C01789=1059.160,245.472,-93.198,172.780,33.846,156.300
C01790=1059.154,245.224,-93.170,172.776,33.843,156.299
C01791=1059.148,244.975,-93.142,172.774,33.838,156.298
C01792=1059.142,244.726,-93.114,172.772,33.835,156.298
C01793=1059.135,244.479,-93.085,172.770,33.831,156.297
C01794=1059.129,244.231,-93.057,172.767,33.827,156.296
C01795=1059.123,243.982,-93.029,172.765,33.823,156.295
C01796=1059.117,243.733,-93.001,172.763,33.820,156.295
C01797=1059.111,243.485,-92.973,172.761,33.816,156.294
C01798=1059.105,243.237,-92.945,172.759,33.812,156.293
C01799=1059.099,242.988,-92.917,172.755,33.808,156.292
C01800=1059.092,242.740,-92.889,172.753,33.804,156.292
C01801=1059.087,242.492,-92.861,172.751,33.801,156.291
C01802=1059.080,242.243,-92.834,172.749,33.797,156.290
C01803=1059.074,241.994,-92.805,172.747,33.793,156.290
C01804=1059.068,241.747,-92.778,172.744,33.789,156.289
C01805=1059.061,241.498,-92.750,172.742,33.786,156.288
C01806=1059.056,241.249,-92.722,172.740,33.782,156.287
C01807=1059.049,241.001,-92.694,172.738,33.778,156.287
C01808=1059.043,240.753,-92.667,172.734,33.774,156.286
C01809=1059.037,240.504,-92.639,172.732,33.770,156.285
C01810=1059.030,240.255,-92.612,172.730,33.767,156.285
C01811=1059.024,240.008,-92.584,172.728,33.763,156.284
C01812=1059.018,239.759,-92.556,172.726,33.759,156.283
C01813=1059.012,239.511,-92.528,172.723,33.755,156.282
C01814=1059.006,239.263,-92.501,172.721,33.752,156.282
C01815=1059.000,239.014,-92.472,172.719,33.748,156.281
C01816=1058.993,238.765,-92.445,172.717,33.744,156.280
C01817=1058.987,238.517,-92.418,172.714,33.740,156.279
C01818=1058.981,238.269,-92.390,172.712,33.737,156.279
C01819=1058.975,238.020,-92.362,172.709,33.733,156.278
C01820=1058.969,237.772,-92.335,172.707,33.729,156.277
C01821=1058.962,237.523,-92.308,172.705,33.725,156.276
C01822=1058.956,237.275,-92.280,172.703,33.721,156.276
C01823=1058.950,237.027,-92.252,172.701,33.718,156.275
C01824=1058.944,236.778,-92.225,172.699,33.714,156.274
C01825=1058.938,236.530,-92.198,172.696,33.710,156.274
C01826=1058.932,236.297,-92.171,172.694,33.707,156.273
C01827=1058.926,236.065,-92.146,172.691,33.703,156.272
C01828=1058.920,235.833,-92.121,172.689,33.700,156.272
C01829=1058.915,235.599,-92.094,172.687,33.696,156.271
C01830=1058.909,235.367,-92.069,172.685,33.692,156.270
C01831=1058.903,235.135,-92.043,172.683,33.689,156.270
C01832=1058.897,234.902,-92.017,172.681,33.685,156.269
C01833=1058.892,234.670,-91.992,172.679,33.681,156.268
C01834=1058.885,234.421,-91.964,172.677,33.678,156.267
C01835=1058.880,234.173,-91.937,172.675,33.674,156.267
C01836=1058.873,233.924,-91.910,172.673,33.670,156.266
C01837=1058.867,233.676,-91.883,172.671,33.666,156.265
C01838=1058.861,233.427,-91.855,172.668,33.663,156.265
C01839=1058.855,233.180,-91.827,172.666,33.659,156.264
C01840=1058.849,232.930,-91.800,172.664,33.655,156.263
C01841=1058.843,232.683,-91.773,172.661,33.651,156.262
C01842=1058.836,232.434,-91.746,172.659,33.647,156.262
C01843=1058.830,232.185,-91.719,172.657,33.644,156.261
C01844=1058.824,231.937,-91.691,172.655,33.639,156.260
C01845=1058.818,231.688,-91.665,172.653,33.636,156.259
C01846=1058.811,231.440,-91.637,172.651,33.632,156.259
C01847=1058.806,231.192,-91.610,172.649,33.629,156.258
C01848=1058.800,230.943,-91.582,172.647,33.624,156.257
C01849=1058.794,230.695,-91.555,172.644,33.621,156.256
C01850=1058.787,230.445,-91.528,172.641,33.617,156.256
C01851=1058.781,230.198,-91.501,172.639,33.613,156.255
C01852=1058.775,229.949,-91.474,172.637,33.609,156.254
C01853=1058.769,229.701,-91.447,172.635,33.605,156.254
C01854=1058.763,229.452,-91.420,172.633,33.601,156.253
C01855=1058.757,229.204,-91.393,172.631,33.598,156.252
C01856=1058.750,228.954,-91.366,172.629,33.594,156.251
C01857=1058.744,228.707,-91.339,172.627,33.590,156.251
C01858=1058.737,228.458,-91.312,172.625,33.587,156.250
C01859=1058.731,228.210,-91.286,172.623,33.582,156.249
C01860=1058.725,227.961,-91.258,172.620,33.579,156.248
C01861=1058.719,227.713,-91.231,172.617,33.575,156.248
C01862=1058.713,227.464,-91.205,172.615,33.571,156.247
C01863=1058.707,227.215,-91.178,172.613,33.567,156.246
C01864=1058.700,226.967,-91.152,172.611,33.564,156.246
C01865=1058.694,226.719,-91.124,172.609,33.560,156.245
C01866=1058.688,226.471,-91.097,172.607,33.556,156.244
C01867=1058.681,226.221,-91.070,172.605,33.552,156.243
C01868=1058.676,225.973,-91.043,172.603,33.548,156.243
C01869=1058.670,225.725,-91.017,172.601,33.545,156.242
C01870=1058.663,225.476,-90.990,172.599,33.540,156.241
C01871=1058.657,225.228,-90.963,172.597,33.537,156.241
C01872=1058.650,224.979,-90.936,172.595,33.533,156.240
C01873=1058.645,224.731,-90.909,172.592,33.529,156.239
C01874=1058.639,224.483,-90.883,172.590,33.525,156.238
C01875=1058.632,224.233,-90.856,172.588,33.522,156.238
C01876=1058.626,223.985,-90.830,172.586,33.517,156.237
C01877=1058.620,223.737,-90.803,172.584,33.514,156.236
C01878=1058.614,223.488,-90.776,172.582,33.510,156.235
C01879=1058.608,223.240,-90.749,172.580,33.506,156.235
C01880=1058.602,222.991,-90.723,172.578,33.502,156.234
C01881=1058.595,222.743,-90.696,172.576,33.499,156.233
C01882=1058.590,222.506,-90.670,172.574,33.495,156.233
C01883=1058.584,222.270,-90.646,172.572,33.491,156.232
C01884=1058.578,222.033,-90.620,172.570,33.488,156.231
C01885=1058.572,221.797,-90.595,172.568,33.484,156.230
C01886=1058.566,221.561,-90.570,172.565,33.480,156.230
C01887=1058.561,221.324,-90.544,172.563,33.476,156.229
C01888=1058.555,221.088,-90.519,172.561,33.472,156.228
C01889=1058.549,220.852,-90.493,172.559,33.469,156.228
C01890=1058.543,220.603,-90.468,172.557,33.465,156.227
C01891=1058.537,220.354,-90.441,172.555,33.461,156.226
C01892=1058.530,220.106,-90.415,172.553,33.458,156.225
C01893=1058.524,219.857,-90.388,172.551,33.453,156.225
C01894=1058.517,219.609,-90.362,172.549,33.450,156.224
C01895=1058.511,219.360,-90.335,172.547,33.446,156.223
C01896=1058.505,219.112,-90.309,172.545,33.442,156.222
C01897=1058.499,218.863,-90.283,172.543,33.438,156.222
C01898=1058.493,218.614,-90.256,172.541,33.435,156.221
C01899=1058.486,218.366,-90.230,172.539,33.430,156.220
C01900=1058.481,218.118,-90.203,172.537,33.427,156.220
C01901=1058.474,217.868,-90.177,172.535,33.423,156.219
C01902=1058.468,217.620,-90.151,172.532,33.419,156.218
C01903=1058.462,217.372,-90.125,172.530,33.415,156.217
C01904=1058.456,217.124,-90.098,172.528,33.411,156.217
C01905=1058.449,216.874,-90.072,172.526,33.407,156.216
C01906=1058.443,216.626,-90.046,172.524,33.404,156.215
C01907=1058.437,216.378,-90.020,172.522,33.400,156.215
C01908=1058.431,216.129,-89.993,172.520,33.396,156.214
C01909=1058.424,215.880,-89.967,172.519,33.392,156.213
C01910=1058.418,215.632,-89.941,172.517,33.388,156.212
C01911=1058.412,215.384,-89.915,172.515,33.384,156.212
C01912=1058.406,215.135,-89.889,172.513,33.380,156.211
C01913=1058.400,214.887,-89.863,172.511,33.376,156.210
C01914=1058.394,214.637,-89.836,172.509,33.373,156.209
C01915=1058.387,214.389,-89.810,172.507,33.368,156.209
C01916=1058.382,214.141,-89.784,172.505,33.365,156.208
C01917=1058.375,213.892,-89.758,172.503,33.361,156.207
C01918=1058.370,213.644,-89.732,172.500,33.357,156.206
C01919=1058.363,213.395,-89.706,172.498,33.353,156.206
C01920=1058.358,213.147,-89.680,172.496,33.349,156.205
C01921=1058.350,212.898,-89.653,172.494,33.345,156.204
C01922=1058.345,212.649,-89.627,172.492,33.341,156.203
C01923=1058.338,212.401,-89.601,172.490,33.337,156.203
C01924=1058.333,212.152,-89.575,172.488,33.334,156.202
C01925=1058.327,211.904,-89.549,172.486,33.329,156.201
C01926=1058.320,211.655,-89.524,172.485,33.326,156.200
C01927=1058.314,211.405,-89.498,172.483,33.321,156.200
C01928=1058.308,211.157,-89.472,172.481,33.318,156.199
C01929=1058.302,210.909,-89.446,172.479,33.313,156.198
C01930=1058.296,210.660,-89.420,172.477,33.310,156.197
C01931=1058.290,210.412,-89.394,172.475,33.306,156.197
C01932=1058.283,210.164,-89.368,172.473,33.302,156.196
C01933=1058.277,209.915,-89.343,172.471,33.298,156.195
C01934=1058.271,209.666,-89.317,172.469,33.294,156.194
C01935=1058.265,209.418,-89.291,172.467,33.290,156.194
C01936=1058.258,209.168,-89.265,172.465,33.287,156.193
C01937=1058.252,208.920,-89.239,172.463,33.282,156.192
C01938=1058.246,208.686,-89.215,172.461,33.279,156.192
C01939=1058.241,208.453,-89.191,172.459,33.275,156.191
C01940=1058.234,208.219,-89.167,172.457,33.271,156.190
C01941=1058.229,207.985,-89.143,172.455,33.268,156.190
C01942=1058.223,207.751,-89.119,172.454,33.264,156.189
C01943=1058.217,207.517,-89.094,172.452,33.260,156.188
C01944=1058.212,207.283,-89.070,172.450,33.257,156.187
C01945=1058.206,207.049,-89.046,172.448,33.253,156.187
C01946=1058.180,205.999,-88.941,172.259,33.165,156.176
C01947=1058.174,205.751,-88.916,172.256,33.162,156.175
C01948=1058.169,205.502,-88.892,172.254,33.159,156.175
C01949=1058.163,205.253,-88.867,172.252,33.156,156.174
C01950=1058.157,205.005,-88.843,172.249,33.153,156.173
C01951=1058.151,204.756,-88.818,172.247,33.150,156.173
C01952=1058.145,204.507,-88.793,172.245,33.147,156.172
C01953=1058.139,204.259,-88.768,172.242,33.144,156.172
C01954=1058.133,204.010,-88.743,172.240,33.140,156.171
C01955=1058.128,203.761,-88.719,172.238,33.138,156.171
C01956=1058.122,203.512,-88.694,172.235,33.135,156.170
C01957=1058.116,203.263,-88.669,172.233,33.132,156.170
C01958=1058.110,203.015,-88.645,172.231,33.128,156.169
C01959=1058.104,202.766,-88.621,172.228,33.125,156.169
C01960=1058.098,202.518,-88.596,172.225,33.122,156.168
C01961=1058.092,202.268,-88.571,172.223,33.120,156.168
C01962=1058.087,202.020,-88.547,172.220,33.116,156.167
C01963=1058.081,201.771,-88.521,172.218,33.113,156.166
C01964=1058.074,201.522,-88.497,172.216,33.110,156.166
C01965=1058.069,201.274,-88.473,172.213,33.107,156.165
C01966=1058.062,201.025,-88.449,172.211,33.104,156.165
C01967=1058.057,200.777,-88.424,172.209,33.101,156.164
C01968=1058.050,200.528,-88.400,172.207,33.099,156.164
C01969=1058.044,200.278,-88.375,172.204,33.095,156.163
C01970=1058.039,200.030,-88.351,172.202,33.093,156.163
C01971=1058.032,199.781,-88.327,172.200,33.090,156.162
C01972=1058.026,199.533,-88.302,172.197,33.087,156.162
C01973=1058.020,199.284,-88.278,172.195,33.084,156.161
C01974=1058.015,199.035,-88.254,172.193,33.081,156.161
C01975=1058.008,198.786,-88.230,172.190,33.078,156.160
C01976=1058.003,198.538,-88.206,172.188,33.075,156.160
C01977=1057.996,198.289,-88.182,172.186,33.072,156.159
C01978=1057.991,198.040,-88.157,172.184,33.069,156.159
C01979=1057.984,197.792,-88.132,172.181,33.066,156.158
C01980=1057.978,197.543,-88.108,172.179,33.063,156.158
C01981=1057.973,197.294,-88.084,172.177,33.061,156.157
C01982=1057.966,197.045,-88.060,172.174,33.057,156.157
C01983=1057.961,196.796,-88.035,172.172,33.054,156.156
C01984=1057.955,196.548,-88.012,172.170,33.052,156.156
C01985=1057.949,196.299,-87.987,172.168,33.048,156.155
C01986=1057.943,196.051,-87.964,172.166,33.046,156.155
C01987=1057.937,195.801,-87.939,172.164,33.043,156.154
C01988=1057.931,195.553,-87.915,172.162,33.040,156.154
C01989=1057.925,195.304,-87.891,172.160,33.037,156.153
C01990=1057.919,195.055,-87.867,172.157,33.034,156.153
C01991=1057.913,194.806,-87.842,172.155,33.031,156.152
C01992=1057.907,194.558,-87.819,172.153,33.028,156.152
C01993=1057.901,194.309,-87.794,172.151,33.025,156.151
C01994=1057.895,194.060,-87.770,172.148,33.022,156.151
C01995=1057.890,193.812,-87.746,172.146,33.019,156.150
C01996=1057.883,193.562,-87.723,172.144,33.017,156.150
C01997=1057.878,193.314,-87.699,172.142,33.014,156.149
C01998=1057.871,193.065,-87.675,172.140,33.010,156.149
C01999=1057.866,192.816,-87.650,172.137,33.008,156.148
C02000=1057.860,192.568,-87.627,172.135,33.005,156.148
C02001=1057.854,192.318,-87.602,172.133,33.002,156.147
C02002=1057.848,192.070,-87.578,172.131,32.999,156.147
C02003=1057.843,191.821,-87.555,172.128,32.996,156.146
C02004=1057.836,191.572,-87.531,172.126,32.993,156.146
C02005=1057.831,191.323,-87.507,172.124,32.990,156.145
C02006=1057.824,191.074,-87.482,172.122,32.987,156.145
C02007=1057.819,190.791,-87.456,172.119,32.984,156.144
C02008=1057.812,190.507,-87.428,172.117,32.980,156.143
C02009=1057.805,190.223,-87.401,172.114,32.977,156.143
C02010=1057.799,189.940,-87.373,172.112,32.974,156.142
C02011=1057.792,189.691,-87.349,172.110,32.971,156.142
C02012=1057.787,189.442,-87.326,172.107,32.968,156.141
C02013=1057.781,189.193,-87.302,172.105,32.965,156.141
C02014=1057.774,188.944,-87.278,172.103,32.963,156.140
C02015=1057.769,188.695,-87.255,172.101,32.959,156.140
C02016=1057.763,188.447,-87.231,172.099,32.957,156.139
C02017=1057.758,188.198,-87.207,172.096,32.954,156.139
C02018=1057.752,187.949,-87.183,172.094,32.951,156.138
C02019=1057.746,187.700,-87.159,172.092,32.948,156.138
C02020=1057.740,187.452,-87.136,172.090,32.945,156.137
C02021=1057.735,187.203,-87.113,172.088,32.942,156.137
C02022=1057.729,186.954,-87.088,172.086,32.939,156.136
C02023=1057.723,186.705,-87.064,172.083,32.936,156.136
C02024=1057.718,186.456,-87.041,172.081,32.933,156.135
C02025=1057.712,186.208,-87.017,172.079,32.931,156.135
C02026=1057.706,185.958,-86.993,172.077,32.928,156.134
C02027=1057.700,185.710,-86.970,172.075,32.925,156.134
C02028=1057.694,185.461,-86.946,172.073,32.922,156.133
C02029=1057.689,185.212,-86.922,172.071,32.919,156.133
C02030=1057.683,184.964,-86.899,172.068,32.916,156.132
C02031=1057.677,184.714,-86.875,172.066,32.913,156.132
C02032=1057.671,184.466,-86.851,172.064,32.910,156.131
C02033=1057.666,184.217,-86.828,172.062,32.908,156.131
C02034=1057.660,183.969,-86.804,172.060,32.905,156.130
C02035=1057.653,183.719,-86.781,172.058,32.902,156.130
C02036=1057.647,183.470,-86.758,172.055,32.899,156.129
C02037=1057.641,183.222,-86.735,172.053,32.897,156.129
C02038=1057.635,182.972,-86.711,172.051,32.894,156.128
C02039=1057.629,182.724,-86.688,172.049,32.891,156.128
C02040=1057.623,182.475,-86.665,172.047,32.889,156.128
C02041=1057.618,182.226,-86.642,172.045,32.886,156.127
C02042=1057.610,181.977,-86.618,172.042,32.883,156.127
C02043=1057.604,181.729,-86.595,172.040,32.880,156.126
C02044=1057.599,181.480,-86.572,172.038,32.878,156.126
C02045=1057.593,181.231,-86.549,172.036,32.875,156.125
C02046=1057.586,180.982,-86.525,172.034,32.872,156.125
C02047=1057.581,180.733,-86.502,172.032,32.869,156.124
C02048=1057.575,180.485,-86.479,172.030,32.867,156.124
C02049=1057.569,180.236,-86.456,172.027,32.864,156.123
C02050=1057.563,179.986,-86.433,172.025,32.862,156.123
C02051=1057.557,179.737,-86.410,172.023,32.858,156.122
C02052=1057.550,179.489,-86.387,172.021,32.856,156.122
C02053=1057.544,179.240,-86.364,172.019,32.853,156.122
C02054=1057.539,178.991,-86.341,172.017,32.851,156.121
C02055=1057.532,178.742,-86.317,172.015,32.848,156.121
C02056=1057.526,178.494,-86.294,172.013,32.845,156.120
C02057=1057.520,178.245,-86.271,172.011,32.842,156.120
C02058=1057.515,177.996,-86.248,172.009,32.840,156.119
C02059=1057.509,177.747,-86.225,172.007,32.837,156.119
C02060=1057.502,177.498,-86.202,172.005,32.834,156.118
C02061=1057.496,177.249,-86.178,172.003,32.831,156.118
C02062=1057.490,177.000,-86.155,172.001,32.829,156.117
C02063=1057.484,176.752,-86.133,171.999,32.826,156.117
C02064=1057.479,176.503,-86.110,171.997,32.823,156.116
C02065=1057.473,176.254,-86.087,171.995,32.821,156.116
C02066=1057.467,176.005,-86.064,171.993,32.818,156.116
C02067=1057.461,175.756,-86.041,171.990,32.815,156.115
C02068=1057.454,175.507,-86.018,171.988,32.812,156.115
C02069=1057.448,175.258,-85.994,171.986,32.810,156.114
C02070=1057.443,175.009,-85.971,171.984,32.807,156.114
C02071=1057.436,174.725,-85.946,171.982,32.804,156.113
C02072=1057.429,174.441,-85.919,171.979,32.801,156.113
C02073=1057.422,174.156,-85.893,171.977,32.798,156.112
C02074=1057.416,173.872,-85.867,171.975,32.795,156.112
C02075=1057.410,173.623,-85.844,171.973,32.792,156.111
C02076=1057.404,173.374,-85.822,171.971,32.789,156.111
C02077=1057.398,173.125,-85.799,171.968,32.786,156.110
C02078=1057.393,172.876,-85.776,171.966,32.784,156.110
C02079=1057.386,172.628,-85.753,171.964,32.781,156.109
C02080=1057.380,172.379,-85.730,171.962,32.778,156.109
C02081=1057.375,172.130,-85.707,171.960,32.776,156.108
C02082=1057.369,171.881,-85.684,171.958,32.773,156.108
C02083=1057.363,171.632,-85.661,171.956,32.770,156.108
C02084=1057.357,171.384,-85.639,171.954,32.768,156.107
C02085=1057.351,171.135,-85.616,171.952,32.765,156.107
C02086=1057.345,170.886,-85.593,171.950,32.762,156.106
C02087=1057.340,170.637,-85.570,171.948,32.760,156.106
C02088=1057.334,170.388,-85.547,171.946,32.757,156.105
C02089=1057.327,170.139,-85.525,171.944,32.754,156.105
C02090=1057.322,169.891,-85.502,171.942,32.751,156.104
C02091=1057.316,169.641,-85.480,171.940,32.749,156.104
C02092=1057.311,169.392,-85.457,171.939,32.746,156.103
C02093=1057.305,169.143,-85.434,171.937,32.744,156.103
C02094=1057.298,168.895,-85.412,171.935,32.740,156.102
C02095=1057.293,168.646,-85.389,171.933,32.738,156.102
C02096=1057.287,168.397,-85.366,171.931,32.735,156.102
C02097=1057.281,168.147,-85.343,171.929,32.733,156.101
C02098=1057.275,167.899,-85.321,171.927,32.730,156.101
C02099=1057.269,167.650,-85.298,171.925,32.727,156.100
C02100=1057.264,167.402,-85.276,171.923,32.724,156.100
C02101=1057.258,167.153,-85.253,171.921,32.722,156.099
C02102=1057.252,166.904,-85.231,171.919,32.719,156.099
C02103=1057.246,166.655,-85.208,171.917,32.716,156.098
C02104=1057.241,166.406,-85.185,171.915,32.713,156.098
C02105=1057.235,166.157,-85.162,171.913,32.711,156.097
C02106=1057.229,165.908,-85.141,171.911,32.708,156.097
C02107=1057.223,165.659,-85.118,171.909,32.706,156.097
C02108=1057.217,165.410,-85.095,171.907,32.702,156.096
C02109=1057.213,165.161,-85.073,171.905,32.700,156.096
C02110=1057.206,164.913,-85.050,171.903,32.697,156.095
C02111=1057.200,164.664,-85.027,171.901,32.695,156.095
C02112=1057.195,164.414,-85.005,171.899,32.692,156.094
C02113=1057.189,164.165,-84.982,171.897,32.689,156.094
C02114=1057.183,163.917,-84.960,171.895,32.686,156.093
C02115=1057.177,163.667,-84.938,171.893,32.684,156.093
C02116=1057.172,163.419,-84.915,171.891,32.681,156.092
C02117=1057.166,163.170,-84.892,171.889,32.678,156.092
C02118=1057.160,162.921,-84.871,171.887,32.675,156.091
C02119=1057.155,162.672,-84.848,171.885,32.673,156.091
C02120=1057.149,162.422,-84.825,171.884,32.670,156.091
C02121=1057.143,162.175,-84.803,171.882,32.668,156.090
C02122=1057.138,161.926,-84.780,171.880,32.665,156.090
C02123=1057.132,161.676,-84.758,171.878,32.662,156.089
C02124=1057.126,161.427,-84.735,171.876,32.659,156.089
C02125=1057.120,161.178,-84.714,171.874,32.657,156.088
C02126=1057.115,160.930,-84.691,171.872,32.654,156.088
C02127=1057.109,160.681,-84.669,171.870,32.651,156.087
C02128=1057.103,160.432,-84.646,171.868,32.648,156.087
C02129=1057.097,160.182,-84.625,171.866,32.646,156.087
C02130=1057.091,159.934,-84.603,171.864,32.643,156.086
C02131=1057.085,159.684,-84.580,171.862,32.641,156.086
C02132=1057.079,159.435,-84.559,171.860,32.638,156.085
C02133=1057.074,159.187,-84.536,171.858,32.636,156.085
C02134=1057.068,158.938,-84.514,171.856,32.633,156.084
C02135=1057.061,158.653,-84.489,171.854,32.630,156.084
C02136=1057.054,158.368,-84.464,171.852,32.627,156.083
C02137=1057.047,158.084,-84.439,171.849,32.624,156.083
C02138=1057.040,157.799,-84.414,171.847,32.621,156.082
C02139=1057.034,157.550,-84.391,171.845,32.619,156.082
C02140=1057.029,157.302,-84.370,171.843,32.616,156.082
C02141=1057.023,157.052,-84.348,171.841,32.614,156.081
C02142=1057.017,156.804,-84.325,171.839,32.611,156.081
C02143=1057.011,156.554,-84.303,171.837,32.608,156.080
C02144=1057.005,156.305,-84.282,171.836,32.606,156.080
C02145=1056.999,156.057,-84.259,171.835,32.603,156.079
C02146=1056.993,155.808,-84.237,171.833,32.601,156.079
C02147=1056.987,155.559,-84.216,171.831,32.598,156.079
C02148=1056.981,155.310,-84.193,171.829,32.595,156.078
C02149=1056.976,155.061,-84.172,171.827,32.593,156.078
C02150=1056.970,154.812,-84.150,171.825,32.590,156.077
C02151=1056.963,154.563,-84.128,171.823,32.588,156.077
C02152=1056.958,154.314,-84.105,171.821,32.585,156.076
C02153=1056.952,154.065,-84.084,171.819,32.583,156.076
C02154=1056.946,153.816,-84.062,171.817,32.580,156.076
C02155=1056.940,153.567,-84.041,171.815,32.577,156.075
C02156=1056.934,153.318,-84.019,171.813,32.575,156.075
C02157=1056.928,153.069,-83.996,171.811,32.572,156.074
C02158=1056.922,152.820,-83.975,171.809,32.570,156.074
C02159=1056.916,152.571,-83.953,171.807,32.567,156.073
C02160=1056.910,152.322,-83.932,171.805,32.564,156.073
C02161=1056.904,152.073,-83.910,171.804,32.562,156.072
C02162=1056.898,151.824,-83.889,171.802,32.559,156.072
C02163=1056.893,151.575,-83.867,171.800,32.557,156.072
C02164=1056.887,151.325,-83.845,171.798,32.554,156.071
C02165=1056.881,151.078,-83.823,171.796,32.552,156.071
C02166=1056.875,150.828,-83.801,171.795,32.549,156.070
C02167=1056.869,150.579,-83.780,171.793,32.546,156.070
C02168=1056.863,150.331,-83.758,171.791,32.544,156.069
C02169=1056.858,150.081,-83.736,171.789,32.541,156.069
C02170=1056.851,149.832,-83.715,171.787,32.539,156.069
C02171=1056.846,149.583,-83.693,171.785,32.536,156.068
C02172=1056.840,149.334,-83.672,171.784,32.533,156.068
C02173=1056.833,149.085,-83.650,171.782,32.531,156.067
C02174=1056.828,148.836,-83.629,171.780,32.528,156.067
C02175=1056.822,148.587,-83.607,171.778,32.526,156.066
C02176=1056.816,148.338,-83.585,171.776,32.523,156.066
C02177=1056.810,148.090,-83.564,171.774,32.521,156.066
C02178=1056.804,147.840,-83.543,171.772,32.518,156.065
C02179=1056.798,147.591,-83.520,171.770,32.516,156.065
C02180=1056.792,147.343,-83.500,171.768,32.513,156.064
C02181=1056.786,147.093,-83.478,171.766,32.511,156.064
C02182=1056.780,146.844,-83.456,171.765,32.508,156.064
C02183=1056.774,146.596,-83.435,171.763,32.506,156.063
C02184=1056.768,146.347,-83.413,171.761,32.503,156.063
C02185=1056.762,146.097,-83.393,171.759,32.500,156.062
C02186=1056.757,145.848,-83.371,171.758,32.498,156.062
C02187=1056.751,145.599,-83.350,171.756,32.496,156.062
C02188=1056.744,145.350,-83.328,171.754,32.493,156.061
C02189=1056.739,145.101,-83.307,171.752,32.491,156.061
C02190=1056.733,144.852,-83.285,171.750,32.488,156.060
C02191=1056.726,144.603,-83.263,171.748,32.485,156.060
C02192=1056.721,144.354,-83.242,171.747,32.483,156.059
C02193=1056.715,144.105,-83.221,171.745,32.480,156.059
C02194=1056.709,143.856,-83.201,171.743,32.478,156.059
C02195=1056.703,143.607,-83.179,171.741,32.476,156.058
C02196=1056.696,143.358,-83.157,171.739,32.473,156.058
C02197=1056.691,143.109,-83.136,171.737,32.470,156.057
C02198=1056.685,142.860,-83.115,171.735,32.468,156.057
C02199=1056.678,142.575,-83.090,171.733,32.465,156.056
C02200=1056.672,142.290,-83.066,171.731,32.462,156.056
C02201=1056.665,142.005,-83.043,171.729,32.459,156.055
C02202=1056.658,141.720,-83.018,171.727,32.456,156.055
C02203=1056.653,141.472,-82.996,171.725,32.454,156.055
C02204=1056.646,141.222,-82.975,171.724,32.451,156.054
C02205=1056.640,140.973,-82.954,171.722,32.448,156.054
C02206=1056.634,140.724,-82.933,171.720,32.446,156.053
C02207=1056.628,140.475,-82.911,171.719,32.444,156.053
C02208=1056.623,140.226,-82.891,171.717,32.441,156.053
C02209=1056.617,139.977,-82.869,171.715,32.439,156.052
C02210=1056.611,139.728,-82.848,171.713,32.436,156.052
C02211=1056.605,139.478,-82.827,171.711,32.434,156.051
C02212=1056.599,139.230,-82.806,171.709,32.431,156.051
C02213=1056.593,138.981,-82.785,171.707,32.428,156.050
C02214=1056.588,138.732,-82.764,171.706,32.426,156.050
C02215=1056.581,138.483,-82.743,171.704,32.424,156.050
C02216=1056.575,138.234,-82.723,171.702,32.421,156.049
C02217=1056.569,137.985,-82.701,171.700,32.419,156.049
C02218=1056.563,137.735,-82.679,171.698,32.416,156.048
C02219=1056.557,137.487,-82.659,171.696,32.413,156.048
C02220=1056.551,137.237,-82.638,171.695,32.411,156.048
C02221=1056.546,136.988,-82.617,171.693,32.409,156.047
C02222=1056.539,136.739,-82.596,171.692,32.406,156.047
C02223=1056.533,136.490,-82.576,171.690,32.404,156.046
C02224=1056.527,136.241,-82.554,171.688,32.401,156.046
C02225=1056.521,135.992,-82.534,171.686,32.398,156.046
C02226=1056.515,135.743,-82.512,171.684,32.396,156.045
C02227=1056.510,135.494,-82.492,171.683,32.394,156.045
C02228=1056.503,135.245,-82.471,171.681,32.391,156.044
C02229=1056.498,134.996,-82.450,171.679,32.389,156.044
C02230=1056.492,134.747,-82.429,171.677,32.386,156.043
C02231=1056.486,134.498,-82.409,171.675,32.384,156.043
C02232=1056.479,134.249,-82.387,171.673,32.381,156.043
C02233=1056.474,134.000,-82.366,171.672,32.379,156.042
C02234=1056.468,133.751,-82.346,171.670,32.376,156.042
C02235=1056.462,133.502,-82.325,171.668,32.374,156.041
C02236=1056.457,133.252,-82.304,171.666,32.371,156.041
C02237=1056.450,133.004,-82.283,171.664,32.369,156.041
C02238=1056.445,132.754,-82.263,171.664,32.367,156.040
C02239=1056.438,132.506,-82.242,171.662,32.364,156.040
C02240=1056.432,132.256,-82.221,171.660,32.361,156.039
C02241=1056.427,132.007,-82.201,171.658,32.359,156.039
C02242=1056.420,131.758,-82.180,171.656,32.356,156.039
C02243=1056.415,131.509,-82.159,171.654,32.354,156.038
C02244=1056.408,131.260,-82.139,171.653,32.352,156.038
C02245=1056.403,131.011,-82.117,171.651,32.349,156.037
C02246=1056.396,130.762,-82.097,171.649,32.347,156.037
C02247=1056.390,130.513,-82.077,171.647,32.344,156.037
C02248=1056.384,130.264,-82.055,171.645,32.342,156.036
C02249=1056.378,130.015,-82.035,171.644,32.340,156.036
C02250=1056.372,129.765,-82.015,171.642,32.337,156.035
C02251=1056.366,129.516,-81.995,171.640,32.335,156.035
C02252=1056.359,129.267,-81.974,171.638,32.332,156.035
C02253=1056.353,129.019,-81.954,171.636,32.330,156.034
C02254=1056.348,128.769,-81.933,171.635,32.327,156.034
C02255=1056.342,128.520,-81.913,171.634,32.325,156.033
C02256=1056.336,128.271,-81.891,171.632,32.323,156.033
C02257=1056.329,128.022,-81.871,171.630,32.320,156.033
C02258=1056.323,127.773,-81.851,171.628,32.318,156.032
C02259=1056.318,127.523,-81.830,171.626,32.315,156.032
C02260=1056.312,127.274,-81.810,171.625,32.313,156.032
C02261=1056.306,127.026,-81.790,171.623,32.311,156.031
C02262=1056.299,126.776,-81.769,171.621,32.308,156.031
C02263=1056.292,126.492,-81.746,171.619,32.305,156.030
C02264=1056.285,126.207,-81.722,171.617,32.303,156.030
C02265=1056.279,125.922,-81.699,171.615,32.300,156.029
C02266=1056.272,125.636,-81.676,171.613,32.297,156.029
C02267=1056.266,125.388,-81.655,171.611,32.295,156.029
C02268=1056.259,125.138,-81.635,171.609,32.292,156.028
C02269=1056.254,124.889,-81.615,171.608,32.290,156.028
C02270=1056.248,124.640,-81.595,171.607,32.287,156.027
C02271=1056.241,124.391,-81.574,171.605,32.285,156.027
C02272=1056.236,124.142,-81.554,171.603,32.282,156.027
C02273=1056.230,123.893,-81.534,171.601,32.280,156.026
C02274=1056.224,123.643,-81.513,171.600,32.277,156.026
C02275=1056.218,123.395,-81.493,171.598,32.275,156.025
C02276=1056.212,123.145,-81.473,171.596,32.273,156.025
C02277=1056.206,122.896,-81.453,171.594,32.270,156.025
C02278=1056.200,122.647,-81.433,171.592,32.268,156.024
C02279=1056.194,122.398,-81.412,171.591,32.265,156.024
C02280=1056.188,122.148,-81.392,171.589,32.263,156.023
C02281=1056.182,121.900,-81.372,171.587,32.260,156.023
C02282=1056.177,121.651,-81.351,171.585,32.258,156.023
C02283=1056.171,121.402,-81.331,171.585,32.256,156.022
C02284=1056.164,121.152,-81.311,171.583,32.253,156.022
C02285=1056.158,120.903,-81.291,171.581,32.250,156.021
C02286=1056.153,120.654,-81.270,171.579,32.248,156.021
C02287=1056.146,120.405,-81.250,171.577,32.246,156.021
C02288=1056.140,120.156,-81.230,171.576,32.243,156.020
C02289=1056.134,119.907,-81.210,171.574,32.241,156.020
C02290=1056.129,119.658,-81.190,171.572,32.238,156.019
C02291=1056.122,119.408,-81.169,171.570,32.236,156.019
C02292=1056.116,119.160,-81.149,171.569,32.234,156.019
C02293=1056.111,118.911,-81.129,171.567,32.231,156.018
C02294=1056.105,118.662,-81.109,171.565,32.228,156.018
C02295=1056.099,118.412,-81.090,171.563,32.226,156.017
C02296=1056.093,118.163,-81.069,171.562,32.224,156.017
C02297=1056.088,117.914,-81.049,171.561,32.221,156.017
C02298=1056.082,117.665,-81.029,171.559,32.218,156.016
C02299=1056.076,117.416,-81.009,171.557,32.216,156.016
C02300=1056.070,117.167,-80.989,171.556,32.214,156.015
C02301=1056.064,116.917,-80.968,171.554,32.211,156.015
C02302=1056.058,116.668,-80.949,171.552,32.209,156.015
C02303=1056.052,116.419,-80.929,171.550,32.206,156.014
C02304=1056.046,116.170,-80.909,171.549,32.204,156.014
C02305=1056.041,115.921,-80.888,171.547,32.202,156.013
C02306=1056.034,115.672,-80.868,171.545,32.199,156.013
C02307=1056.028,115.422,-80.849,171.543,32.196,156.013
C02308=1056.022,115.173,-80.829,171.542,32.194,156.012
C02309=1056.016,114.925,-80.809,171.540,32.192,156.012
C02310=1056.011,114.676,-80.788,171.538,32.189,156.011
C02311=1056.006,114.426,-80.769,171.538,32.187,156.011
C02312=1056.000,114.177,-80.749,171.536,32.184,156.011
C02313=1055.993,113.928,-80.729,171.534,32.181,156.010
C02314=1055.987,113.679,-80.709,171.532,32.179,156.010
C02315=1055.981,113.430,-80.689,171.531,32.177,156.009
C02316=1055.975,113.181,-80.670,171.529,32.174,156.009
C02317=1055.969,112.932,-80.650,171.527,32.172,156.009
C02318=1055.963,112.682,-80.630,171.525,32.169,156.008
C02319=1055.957,112.433,-80.610,171.524,32.167,156.008
C02320=1055.951,112.184,-80.590,171.522,32.165,156.008
C02321=1055.945,111.935,-80.571,171.520,32.162,156.007
C02322=1055.939,111.686,-80.551,171.518,32.160,156.007
C02323=1055.933,111.437,-80.531,171.517,32.158,156.006
C02324=1055.927,111.187,-80.511,171.516,32.155,156.006
C02325=1055.921,110.938,-80.491,171.514,32.153,156.006
C02326=1055.915,110.689,-80.472,171.512,32.150,156.005
C02327=1055.908,110.404,-80.449,171.510,32.147,156.005
C02328=1055.902,110.118,-80.426,171.508,32.145,156.004
C02329=1055.895,109.833,-80.404,171.506,32.142,156.004
C02330=1055.888,109.548,-80.382,171.505,32.139,156.003
C02331=1055.882,109.300,-80.363,171.503,32.137,156.003
C02332=1055.876,109.049,-80.343,171.501,32.135,156.003
C02333=1055.870,108.801,-80.323,171.499,32.132,156.002
C02334=1055.863,108.551,-80.304,171.498,32.130,156.002
C02335=1055.857,108.303,-80.284,171.496,32.128,156.002
C02336=1055.851,108.053,-80.265,171.495,32.125,156.001
C02337=1055.845,107.804,-80.245,171.493,32.123,156.001
C02338=1055.840,107.555,-80.226,171.492,32.120,156.000
C02339=1055.833,107.305,-80.206,171.490,32.118,156.000
C02340=1055.827,107.056,-80.187,171.488,32.116,156.000
C02341=1055.821,106.807,-80.167,171.486,32.113,155.999
C02342=1055.815,106.558,-80.148,171.485,32.111,155.999
C02343=1055.809,106.309,-80.128,171.483,32.109,155.998
C02344=1055.803,106.060,-80.109,171.481,32.106,155.998
C02345=1055.797,105.811,-80.089,171.480,32.103,155.998
C02346=1055.791,105.562,-80.070,171.478,32.101,155.997
C02347=1055.785,105.312,-80.051,171.476,32.099,155.997
C02348=1055.779,105.064,-80.031,171.474,32.096,155.996
C02349=1055.774,104.814,-80.011,171.474,32.094,155.996
C02350=1055.767,104.566,-79.992,171.472,32.092,155.996
C02351=1055.761,104.316,-79.973,171.470,32.089,155.995
C02352=1055.755,104.067,-79.954,171.469,32.087,155.995
C02353=1055.749,103.817,-79.933,171.467,32.084,155.995
C02354=1055.743,103.568,-79.914,171.465,32.082,155.994
C02355=1055.737,103.319,-79.895,171.463,32.080,155.994
C02356=1055.731,103.070,-79.875,171.462,32.077,155.993
C02357=1055.725,102.821,-79.856,171.460,32.075,155.993
C02358=1055.719,102.571,-79.837,171.458,32.072,155.993
C02359=1055.713,102.322,-79.817,171.457,32.070,155.992
C02360=1055.707,102.073,-79.798,171.455,32.067,155.992
C02361=1055.701,101.824,-79.779,171.454,32.065,155.992
C02362=1055.695,101.575,-79.759,171.453,32.063,155.991
C02363=1055.690,101.325,-79.740,171.451,32.060,155.991
C02364=1055.683,101.076,-79.721,171.449,32.058,155.990
C02365=1055.678,100.827,-79.702,171.447,32.055,155.990
C02366=1055.672,100.578,-79.682,171.446,32.053,155.990
C02367=1055.665,100.329,-79.663,171.444,32.051,155.989
C02368=1055.659,100.080,-79.644,171.442,32.048,155.989
C02369=1055.654,99.830,-79.625,171.441,32.046,155.988
C02370=1055.647,99.581,-79.606,171.439,32.044,155.988
C02371=1055.641,99.332,-79.586,171.437,32.041,155.988
C02372=1055.635,99.083,-79.568,171.435,32.039,155.987
C02373=1055.629,98.834,-79.548,171.435,32.036,155.987
C02374=1055.623,98.585,-79.530,171.433,32.034,155.987
C02375=1055.617,98.335,-79.511,171.431,32.032,155.986
C02376=1055.611,98.086,-79.492,171.430,32.029,155.986
C02377=1055.605,97.837,-79.472,171.428,32.027,155.985
C02378=1055.598,97.588,-79.453,171.426,32.025,155.985
C02379=1055.593,97.339,-79.434,171.424,32.022,155.985
C02380=1055.586,97.089,-79.415,171.423,32.020,155.984
C02381=1055.580,96.840,-79.396,171.421,32.018,155.984
C02382=1055.575,96.591,-79.377,171.419,32.015,155.984
C02383=1055.568,96.341,-79.358,171.418,32.013,155.983
C02384=1055.563,96.092,-79.339,171.417,32.011,155.983
C02385=1055.556,95.843,-79.320,171.415,32.008,155.982
C02386=1055.551,95.593,-79.301,171.414,32.006,155.982
C02387=1055.544,95.344,-79.282,171.412,32.004,155.982
C02388=1055.538,95.096,-79.262,171.410,32.001,155.981
C02389=1055.532,94.847,-79.244,171.408,31.999,155.981
C02390=1055.527,94.598,-79.225,171.407,31.996,155.981
C02391=1055.520,94.312,-79.204,171.405,31.994,155.980
C02392=1055.512,94.027,-79.182,171.403,31.991,155.980
C02393=1055.506,93.742,-79.160,171.401,31.988,155.979
C02394=1055.499,93.457,-79.139,171.399,31.986,155.979
C02395=1055.493,93.207,-79.120,171.398,31.983,155.978
C02396=1055.487,92.958,-79.101,171.397,31.981,155.978
C02397=1055.481,92.709,-79.083,171.395,31.978,155.978
C02398=1055.475,92.460,-79.063,171.393,31.976,155.977
C02399=1055.468,92.211,-79.045,171.392,31.973,155.977
C02400=1055.463,91.961,-79.025,171.390,31.971,155.977
C02401=1055.456,91.712,-79.007,171.388,31.969,155.976
C02402=1055.451,91.463,-78.988,171.387,31.967,155.976
C02403=1055.445,91.214,-78.969,171.385,31.964,155.975
C02404=1055.439,90.965,-78.950,171.383,31.961,155.975
C02405=1055.433,90.716,-78.931,171.382,31.959,155.975
C02406=1055.427,90.466,-78.912,171.381,31.957,155.974
C02407=1055.421,90.217,-78.893,171.379,31.955,155.974
C02408=1055.414,89.967,-78.876,171.377,31.952,155.974
C02409=1055.409,89.718,-78.856,171.376,31.950,155.973
C02410=1055.402,89.469,-78.838,171.374,31.948,155.973
C02411=1055.396,89.220,-78.819,171.372,31.945,155.972
C02412=1055.390,88.971,-78.801,171.371,31.943,155.972
C02413=1055.384,88.722,-78.781,171.369,31.940,155.972
C02414=1055.378,88.472,-78.764,171.367,31.938,155.971
C02415=1055.372,88.223,-78.745,171.366,31.936,155.971
C02416=1055.365,87.974,-78.726,171.364,31.934,155.971
C02417=1055.359,87.725,-78.708,171.363,31.931,155.970
C02418=1055.353,87.475,-78.688,171.361,31.929,155.970
C02419=1055.347,87.225,-78.670,171.360,31.926,155.969
C02420=1055.341,86.977,-78.652,171.358,31.924,155.969
C02421=1055.335,86.728,-78.633,171.356,31.922,155.969
C02422=1055.329,86.479,-78.614,171.355,31.920,155.968
C02423=1055.323,86.229,-78.596,171.353,31.917,155.968
C02424=1055.317,85.980,-78.578,171.351,31.915,155.968
C02425=1055.310,85.731,-78.559,171.350,31.913,155.967
C02426=1055.304,85.482,-78.541,171.348,31.910,155.967
C02427=1055.299,85.232,-78.522,171.346,31.908,155.967
C02428=1055.293,84.983,-78.504,171.346,31.905,155.966
C02429=1055.286,84.734,-78.485,171.344,31.903,155.966
C02430=1055.280,84.484,-78.467,171.342,31.901,155.965
C02431=1055.274,84.235,-78.448,171.341,31.899,155.965
C02432=1055.269,83.986,-78.429,171.339,31.896,155.965
C02433=1055.262,83.736,-78.411,171.337,31.894,155.964
C02434=1055.256,83.487,-78.393,171.336,31.891,155.964
C02435=1055.250,83.238,-78.374,171.334,31.889,155.964
C02436=1055.244,82.989,-78.357,171.332,31.887,155.963
C02437=1055.238,82.740,-78.337,171.331,31.884,155.963
C02438=1055.232,82.491,-78.319,171.330,31.882,155.962
C02439=1055.226,82.241,-78.301,171.328,31.879,155.962
C02440=1055.219,81.992,-78.282,171.327,31.878,155.962
C02441=1055.214,81.743,-78.265,171.325,31.875,155.961
C02442=1055.208,81.493,-78.245,171.323,31.873,155.961
C02443=1055.202,81.244,-78.227,171.321,31.870,155.961
C02444=1055.196,80.994,-78.209,171.320,31.868,155.960
C02445=1055.190,80.746,-78.190,171.318,31.866,155.960
C02446=1055.184,80.496,-78.173,171.316,31.863,155.959
C02447=1055.177,80.247,-78.154,171.315,31.861,155.959
C02448=1055.173,79.998,-78.136,171.313,31.858,155.959
C02449=1055.166,79.749,-78.117,171.312,31.856,155.958
C02450=1055.160,79.499,-78.099,171.311,31.854,155.958
C02451=1055.154,79.250,-78.080,171.309,31.851,155.958
C02452=1055.148,79.001,-78.062,171.307,31.849,155.957
C02453=1055.142,78.752,-78.044,171.306,31.846,155.957
C02454=1055.135,78.503,-78.026,171.304,31.844,155.957
C02455=1055.129,78.218,-78.005,171.302,31.842,155.956
C02456=1055.122,77.932,-77.984,171.300,31.839,155.956
C02457=1055.115,77.647,-77.963,171.298,31.836,155.955
C02458=1055.108,77.361,-77.942,171.297,31.834,155.955
C02459=1055.102,77.112,-77.924,171.296,31.831,155.954
C02460=1055.096,76.864,-77.907,171.294,31.829,155.954
C02461=1055.089,76.614,-77.889,171.292,31.827,155.954
C02462=1055.083,76.364,-77.871,171.291,31.825,155.953
C02463=1055.077,76.116,-77.852,171.289,31.822,155.953
C02464=1055.071,75.866,-77.834,171.287,31.820,155.953
C02465=1055.065,75.617,-77.816,171.286,31.817,155.952
C02466=1055.059,75.367,-77.798,171.284,31.815,155.952
C02467=1055.053,75.118,-77.780,171.282,31.813,155.952
C02468=1055.047,74.869,-77.762,171.282,31.811,155.951
C02469=1055.041,74.619,-77.744,171.280,31.808,155.951
C02470=1055.035,74.370,-77.726,171.278,31.806,155.951
C02471=1055.029,74.121,-77.707,171.277,31.803,155.950
C02472=1055.023,73.871,-77.690,171.275,31.801,155.950
C02473=1055.017,73.622,-77.672,171.273,31.799,155.949
C02474=1055.010,73.373,-77.654,171.272,31.797,155.949
C02475=1055.004,73.124,-77.636,171.270,31.794,155.949
C02476=1054.998,72.875,-77.618,171.268,31.792,155.948
C02477=1054.992,72.626,-77.600,171.267,31.789,155.948
C02478=1054.986,72.376,-77.582,171.266,31.787,155.948
C02479=1054.980,72.127,-77.564,171.264,31.785,155.947
C02480=1054.974,71.877,-77.546,171.263,31.783,155.947
C02481=1054.968,71.629,-77.528,171.261,31.780,155.947
C02482=1054.962,71.379,-77.510,171.259,31.778,155.946
C02483=1054.955,71.129,-77.493,171.258,31.776,155.946
C02484=1054.950,70.880,-77.475,171.256,31.773,155.945
C02485=1054.943,70.631,-77.457,171.254,31.771,155.945
C02486=1054.937,70.381,-77.439,171.253,31.769,155.945
C02487=1054.932,70.132,-77.421,171.251,31.766,155.944
C02488=1054.926,69.883,-77.403,171.250,31.764,155.944
C02489=1054.920,69.634,-77.386,171.249,31.762,155.944
C02490=1054.913,69.385,-77.368,171.247,31.760,155.943
C02491=1054.907,69.135,-77.350,171.245,31.757,155.943
C02492=1054.901,68.886,-77.332,171.244,31.755,155.943
C02493=1054.895,68.636,-77.314,171.242,31.752,155.942
C02494=1054.889,68.388,-77.297,171.240,31.750,155.942
C02495=1054.883,68.138,-77.279,171.239,31.748,155.942
C02496=1054.876,67.889,-77.261,171.237,31.746,155.941
C02497=1054.870,67.640,-77.244,171.236,31.744,155.941
C02498=1054.864,67.390,-77.226,171.235,31.741,155.940
C02499=1054.858,67.141,-77.208,171.233,31.739,155.940
C02500=1054.852,66.891,-77.190,171.231,31.736,155.940
C02501=1054.846,66.642,-77.173,171.230,31.734,155.939
C02502=1054.840,66.393,-77.155,171.228,31.732,155.939
C02503=1054.834,66.143,-77.137,171.226,31.730,155.939
C02504=1054.828,65.895,-77.120,171.224,31.727,155.938
C02505=1054.822,65.645,-77.102,171.223,31.725,155.938
C02506=1054.816,65.396,-77.085,171.221,31.723,155.938
C02507=1054.809,65.146,-77.067,171.220,31.720,155.937
C02508=1054.803,64.897,-77.050,171.219,31.718,155.937
C02509=1054.797,64.648,-77.032,171.217,31.716,155.937
C02510=1054.791,64.398,-77.015,171.215,31.714,155.936
C02511=1054.785,64.149,-76.997,171.214,31.711,155.936
C02512=1054.779,63.899,-76.979,171.212,31.709,155.936
C02513=1054.773,63.651,-76.962,171.210,31.707,155.935
C02514=1054.766,63.401,-76.945,171.209,31.704,155.935
C02515=1054.760,63.151,-76.927,171.207,31.702,155.934
C02516=1054.753,62.903,-76.910,171.206,31.700,155.934
C02517=1054.747,62.653,-76.892,171.205,31.698,155.934
C02518=1054.741,62.404,-76.875,171.203,31.696,155.933
C02519=1054.734,62.118,-76.855,171.201,31.693,155.933
C02520=1054.726,61.833,-76.835,171.199,31.690,155.933
C02521=1054.720,61.548,-76.815,171.197,31.688,155.932
C02522=1054.713,61.263,-76.795,171.195,31.685,155.932
C02523=1054.706,61.013,-76.778,171.194,31.683,155.932
C02524=1054.700,60.764,-76.761,171.192,31.681,155.931
C02525=1054.694,60.514,-76.743,171.191,31.679,155.931
C02526=1054.687,60.266,-76.726,171.190,31.677,155.931
C02527=1054.681,60.016,-76.708,171.188,31.674,155.930
C02528=1054.675,59.767,-76.691,171.186,31.672,155.930
C02529=1054.669,59.517,-76.673,171.184,31.669,155.929
C02530=1054.663,59.268,-76.657,171.183,31.667,155.929
C02531=1054.656,59.019,-76.640,171.181,31.665,155.929
C02532=1054.650,58.770,-76.622,171.179,31.663,155.928
C02533=1054.644,58.520,-76.605,171.178,31.661,155.928
C02534=1054.638,58.271,-76.587,171.177,31.659,155.928
C02535=1054.632,58.021,-76.571,171.175,31.656,155.927
C02536=1054.625,57.772,-76.554,171.174,31.654,155.927
C02537=1054.619,57.523,-76.536,171.172,31.652,155.927
C02538=1054.613,57.274,-76.519,171.170,31.649,155.926
C02539=1054.607,57.024,-76.501,171.169,31.647,155.926
C02540=1054.601,56.775,-76.485,171.167,31.645,155.926
C02541=1054.594,56.525,-76.467,171.165,31.643,155.925
C02542=1054.588,56.276,-76.450,171.164,31.641,155.925
C02543=1054.582,56.027,-76.432,171.163,31.639,155.925
C02544=1054.576,55.777,-76.416,171.161,31.636,155.924
C02545=1054.570,55.528,-76.399,171.160,31.634,155.924
C02546=1054.563,55.279,-76.381,171.158,31.631,155.924
C02547=1054.558,55.029,-76.364,171.156,31.629,155.923
C02548=1054.551,54.780,-76.347,171.154,31.627,155.923
C02549=1054.545,54.531,-76.330,171.153,31.625,155.923
C02550=1054.539,54.281,-76.313,171.151,31.622,155.922
C02551=1054.533,54.032,-76.296,171.149,31.620,155.922
C02552=1054.527,53.783,-76.278,171.149,31.618,155.922
C02553=1054.521,53.533,-76.262,171.147,31.616,155.921
C02554=1054.515,53.284,-76.245,171.145,31.613,155.921
C02555=1054.508,53.035,-76.227,171.144,31.611,155.921
C02556=1054.502,52.785,-76.211,171.142,31.609,155.920
C02557=1054.496,52.536,-76.194,171.140,31.606,155.920
C02558=1054.490,52.287,-76.176,171.139,31.604,155.920
C02559=1054.484,52.037,-76.159,171.137,31.602,155.919
C02560=1054.478,51.789,-76.142,171.136,31.600,155.919
C02561=1054.472,51.538,-76.125,171.135,31.598,155.919
C02562=1054.466,51.290,-76.108,171.133,31.595,155.918
C02563=1054.459,51.040,-76.091,171.131,31.593,155.918
C02564=1054.454,50.790,-76.074,171.130,31.591,155.918
C02565=1054.448,50.542,-76.057,171.128,31.588,155.917
C02566=1054.441,50.292,-76.040,171.126,31.586,155.917
C02567=1054.435,50.043,-76.023,171.125,31.584,155.916
C02568=1054.429,49.793,-76.007,171.123,31.582,155.916
C02569=1054.423,49.544,-75.989,171.122,31.580,155.916
C02570=1054.417,49.294,-75.972,171.121,31.577,155.915
C02571=1054.411,49.045,-75.955,171.119,31.575,155.915
C02572=1054.405,48.795,-75.939,171.117,31.572,155.915
C02573=1054.399,48.546,-75.921,171.116,31.570,155.914
C02574=1054.393,48.297,-75.905,171.114,31.568,155.914
C02575=1054.387,48.048,-75.888,171.112,31.565,155.914
C02576=1054.381,47.798,-75.871,171.111,31.564,155.913
C02577=1054.375,47.549,-75.854,171.110,31.561,155.913
C02578=1054.369,47.300,-75.838,171.108,31.559,155.913
C02579=1054.363,47.050,-75.820,171.106,31.557,155.912
C02580=1054.357,46.801,-75.803,171.105,31.554,155.912
C02581=1054.351,46.552,-75.786,171.103,31.552,155.912
C02582=1054.345,46.303,-75.770,171.101,31.549,155.911
C02583=1054.338,46.017,-75.750,171.100,31.547,155.911
C02584=1054.332,45.731,-75.731,171.098,31.544,155.910
C02585=1054.324,45.445,-75.712,171.096,31.542,155.910
C02586=1054.317,45.160,-75.692,171.095,31.539,155.910
C02587=1054.311,44.910,-75.676,171.093,31.537,155.909
C02588=1054.305,44.661,-75.659,171.091,31.535,155.909
C02589=1054.299,44.412,-75.642,171.090,31.532,155.909
C02590=1054.294,44.162,-75.626,171.088,31.530,155.908
C02591=1054.287,43.913,-75.608,171.086,31.528,155.908
C02592=1054.281,43.664,-75.592,171.085,31.525,155.908
C02593=1054.275,43.414,-75.576,171.083,31.523,155.907
C02594=1054.269,43.165,-75.558,171.082,31.520,155.907
C02595=1054.263,42.915,-75.542,171.081,31.519,155.907
C02596=1054.257,42.666,-75.525,171.079,31.516,155.906
C02597=1054.250,42.417,-75.508,171.077,31.514,155.906
C02598=1054.245,42.168,-75.492,171.076,31.512,155.906
C02599=1054.238,41.918,-75.476,171.074,31.510,155.905
C02600=1054.232,41.668,-75.459,171.072,31.508,155.905
C02601=1054.226,41.420,-75.442,171.070,31.505,155.905
C02602=1054.220,41.170,-75.426,171.070,31.503,155.904
C02603=1054.213,40.920,-75.409,171.068,31.501,155.904
C02604=1054.207,40.671,-75.393,171.066,31.498,155.904
C02605=1054.201,40.422,-75.376,171.065,31.496,155.903
C02606=1054.195,40.173,-75.360,171.063,31.494,155.903
C02607=1054.189,39.923,-75.343,171.061,31.492,155.903
C02608=1054.183,39.673,-75.327,171.060,31.490,155.902
C02609=1054.177,39.424,-75.311,171.058,31.487,155.902
C02610=1054.170,39.175,-75.294,171.057,31.485,155.902
C02611=1054.164,38.926,-75.278,171.056,31.483,155.901
C02612=1054.158,38.676,-75.261,171.054,31.481,155.901
C02613=1054.152,38.426,-75.245,171.052,31.479,155.901
C02614=1054.146,38.177,-75.228,171.050,31.476,155.900
C02615=1054.141,37.927,-75.212,171.049,31.474,155.900
C02616=1054.134,37.679,-75.195,171.047,31.472,155.900
C02617=1054.128,37.430,-75.179,171.045,31.470,155.899
C02618=1054.121,37.180,-75.162,171.045,31.467,155.899
C02619=1054.115,36.930,-75.146,171.043,31.465,155.899
C02620=1054.109,36.681,-75.130,171.041,31.463,155.898
C02621=1054.103,36.432,-75.114,171.040,31.461,155.898
C02622=1054.097,36.182,-75.097,171.038,31.459,155.898
C02623=1054.090,35.933,-75.081,171.036,31.456,155.897
C02624=1054.084,35.683,-75.065,171.034,31.454,155.897
C02625=1054.078,35.434,-75.049,171.033,31.452,155.897
C02626=1054.072,35.184,-75.033,171.032,31.450,155.896
C02627=1054.066,34.935,-75.016,171.030,31.448,155.896
C02628=1054.060,34.685,-75.000,171.029,31.445,155.896
C02629=1054.053,34.436,-74.984,171.027,31.443,155.895
C02630=1054.047,34.187,-74.968,171.025,31.441,155.895
C02631=1054.041,33.937,-74.951,171.023,31.439,155.895
C02632=1054.035,33.688,-74.935,171.022,31.437,155.894
C02633=1054.029,33.439,-74.919,171.020,31.435,155.894
C02634=1054.022,33.189,-74.903,171.019,31.432,155.894
C02635=1054.016,32.940,-74.887,171.018,31.431,155.894
C02636=1054.010,32.690,-74.870,171.016,31.428,155.893
C02637=1054.004,32.441,-74.854,171.014,31.426,155.893
C02638=1053.998,32.192,-74.838,171.012,31.424,155.893
C02639=1053.992,31.942,-74.822,171.011,31.422,155.892
C02640=1053.986,31.693,-74.806,171.009,31.420,155.892
C02641=1053.980,31.444,-74.790,171.007,31.417,155.892
C02642=1053.974,31.194,-74.773,171.007,31.415,155.891
C02643=1053.967,30.944,-74.757,171.005,31.413,155.891
C02644=1053.960,30.695,-74.741,171.003,31.411,155.891
C02645=1053.955,30.446,-74.725,171.001,31.409,155.890
C02646=1053.949,30.197,-74.709,171.000,31.406,155.890
C02647=1053.942,29.911,-74.690,170.998,31.404,155.890
C02648=1053.935,29.626,-74.672,170.996,31.401,155.889
C02649=1053.928,29.339,-74.654,170.994,31.399,155.889
C02650=1053.921,29.054,-74.635,170.993,31.396,155.889
C02651=1053.915,28.804,-74.619,170.991,31.394,155.888
C02652=1053.908,28.555,-74.603,170.989,31.392,155.888
C02653=1053.902,28.305,-74.588,170.988,31.390,155.888
C02654=1053.897,28.056,-74.572,170.986,31.388,155.887
C02655=1053.890,27.807,-74.556,170.984,31.385,155.887
C02656=1053.884,27.558,-74.540,170.983,31.384,155.887
C02657=1053.877,27.309,-74.524,170.982,31.381,155.886
C02658=1053.871,27.058,-74.508,170.980,31.379,155.886
C02659=1053.865,26.809,-74.492,170.978,31.377,155.886
C02660=1053.858,26.560,-74.476,170.977,31.375,155.885
C02661=1053.852,26.310,-74.460,170.975,31.373,155.885
C02662=1053.847,26.060,-74.444,170.973,31.370,155.885
C02663=1053.840,25.811,-74.429,170.971,31.368,155.884
C02664=1053.834,25.562,-74.412,170.970,31.366,155.884
C02665=1053.827,25.313,-74.397,170.969,31.364,155.884
C02666=1053.822,25.063,-74.381,170.967,31.362,155.883
C02667=1053.815,24.814,-74.366,170.966,31.360,155.883
C02668=1053.809,24.565,-74.349,170.964,31.358,155.883
C02669=1053.803,24.315,-74.334,170.962,31.355,155.883
C02670=1053.797,24.066,-74.318,170.960,31.353,155.882
C02671=1053.791,23.816,-74.302,170.959,31.351,155.882
C02672=1053.784,23.567,-74.287,170.957,31.349,155.882
C02673=1053.778,23.317,-74.271,170.956,31.347,155.881
C02674=1053.772,23.068,-74.255,170.954,31.344,155.881
C02675=1053.766,22.818,-74.239,170.953,31.343,155.881
C02676=1053.759,22.569,-74.224,170.951,31.340,155.880
C02677=1053.754,22.320,-74.207,170.949,31.338,155.880
C02678=1053.747,22.070,-74.193,170.947,31.336,155.880
C02679=1053.741,21.821,-74.176,170.946,31.334,155.880
C02680=1053.736,21.571,-74.161,170.944,31.332,155.879
C02681=1053.729,21.322,-74.145,170.943,31.329,155.879
C02682=1053.723,21.072,-74.129,170.942,31.327,155.879
C02683=1053.717,20.823,-74.114,170.940,31.325,155.878
C02684=1053.711,20.573,-74.098,170.938,31.323,155.878
C02685=1053.704,20.324,-74.083,170.936,31.321,155.878
C02686=1053.698,20.074,-74.066,170.935,31.319,155.877
C02687=1053.692,19.825,-74.051,170.933,31.317,155.877
C02688=1053.686,19.575,-74.035,170.931,31.315,155.877
C02689=1053.679,19.326,-74.020,170.930,31.313,155.876
C02690=1053.673,19.077,-74.005,170.929,31.311,155.876
C02691=1053.667,18.827,-73.988,170.927,31.309,155.876
C02692=1053.660,18.578,-73.973,170.925,31.307,155.876
C02693=1053.655,18.328,-73.957,170.923,31.304,155.875
C02694=1053.648,18.079,-73.942,170.922,31.302,155.875
C02695=1053.641,17.830,-73.927,170.920,31.300,155.875
C02696=1053.636,17.580,-73.911,170.919,31.298,155.874
C02697=1053.630,17.331,-73.896,170.917,31.296,155.874
C02698=1053.624,17.081,-73.880,170.916,31.294,155.874
C02699=1053.618,16.832,-73.865,170.914,31.292,155.873
C02700=1053.611,16.583,-73.850,170.912,31.290,155.873
C02701=1053.605,16.333,-73.834,170.910,31.287,155.873
C02702=1053.599,16.084,-73.818,170.909,31.285,155.873
C02703=1053.593,15.834,-73.803,170.907,31.283,155.872
C02704=1053.587,15.584,-73.788,170.906,31.281,155.872
C02705=1053.580,15.335,-73.772,170.904,31.279,155.872
C02706=1053.574,15.085,-73.757,170.903,31.277,155.871
C02707=1053.568,14.837,-73.741,170.901,31.275,155.871
C02708=1053.562,14.587,-73.726,170.899,31.273,155.871
C02709=1053.556,14.337,-73.711,170.897,31.271,155.871
C02710=1053.550,14.088,-73.695,170.895,31.269,155.870
C02711=1053.542,13.781,-73.677,170.894,31.266,155.870
C02712=1053.534,13.475,-73.658,170.892,31.263,155.869
C02713=1053.526,13.170,-73.639,170.890,31.261,155.869
C02714=1053.518,12.863,-73.621,170.888,31.258,155.869
C02715=1053.512,12.624,-73.606,170.886,31.256,155.868
C02716=1053.507,12.386,-73.592,170.884,31.255,155.868
C02717=1053.501,12.147,-73.577,170.883,31.253,155.868
C02718=1053.494,11.909,-73.562,170.882,31.251,155.868
C02719=1053.489,11.671,-73.548,170.880,31.249,155.867
C02720=1053.482,11.432,-73.533,170.879,31.247,155.867
C02721=1053.476,11.193,-73.519,170.877,31.245,155.867
C02722=1053.470,10.955,-73.504,170.875,31.243,155.867
C02723=1053.464,10.705,-73.489,170.873,31.241,155.866
C02724=1053.458,10.456,-73.474,170.872,31.239,155.866
C02725=1053.452,10.206,-73.459,170.870,31.237,155.866
C02726=1053.445,9.957,-73.444,170.869,31.235,155.865
C02727=1053.439,9.707,-73.429,170.867,31.233,155.865
C02728=1053.433,9.458,-73.414,170.865,31.231,155.865
C02729=1053.426,9.208,-73.399,170.864,31.229,155.865
C02730=1053.420,8.959,-73.384,170.862,31.226,155.864
C02731=1053.415,8.709,-73.369,170.860,31.225,155.864
C02732=1053.408,8.460,-73.353,170.858,31.223,155.864
C02733=1053.402,8.210,-73.338,170.857,31.221,155.864
C02734=1053.395,7.961,-73.323,170.856,31.219,155.863
C02735=1053.389,7.711,-73.308,170.854,31.217,155.863
C02736=1053.383,7.462,-73.293,170.852,31.215,155.863
C02737=1053.377,7.213,-73.279,170.850,31.212,155.862
C02738=1053.370,6.963,-73.264,170.849,31.210,155.862
C02739=1053.364,6.714,-73.248,170.847,31.208,155.862
C02740=1053.358,6.464,-73.232,170.845,31.206,155.862
C02741=1053.352,6.215,-73.218,170.844,31.204,155.861
C02742=1053.346,5.965,-73.203,170.842,31.202,155.861
C02743=1053.339,5.716,-73.188,170.841,31.200,155.861
C02744=1053.333,5.466,-73.173,170.839,31.198,155.860
C02745=1053.327,5.217,-73.158,170.837,31.196,155.860
C02746=1053.321,4.967,-73.143,170.835,31.194,155.860
C02747=1053.314,4.718,-73.129,170.834,31.192,155.860
C02748=1053.308,4.468,-73.114,170.833,31.190,155.859
C02749=1053.302,4.219,-73.099,170.831,31.188,155.859
C02750=1053.296,3.969,-73.084,170.829,31.186,155.859
C02751=1053.290,3.719,-73.068,170.827,31.184,155.858
C02752=1053.284,3.470,-73.054,170.826,31.182,155.858
C02753=1053.278,3.221,-73.039,170.824,31.180,155.858
C02754=1053.272,2.971,-73.024,170.822,31.178,155.858
C02755=1053.265,2.722,-73.009,170.820,31.176,155.857
C02756=1053.260,2.473,-72.994,170.819,31.174,155.857
C02757=1053.253,2.223,-72.980,170.818,31.172,155.857
C02758=1053.247,1.973,-72.965,170.816,31.170,155.857
C02759=1053.240,1.724,-72.950,170.814,31.168,155.856
C02760=1053.235,1.475,-72.935,170.812,31.166,155.856
C02761=1053.228,1.225,-72.920,170.810,31.164,155.856
C02762=1053.222,0.975,-72.905,170.809,31.162,155.855
C02763=1053.216,0.726,-72.891,170.808,31.159,155.855
C02764=1053.210,0.477,-72.876,170.806,31.157,155.855
C02765=1053.203,0.227,-72.861,170.804,31.155,155.854
C02766=1053.198,-0.022,-72.846,170.802,31.153,155.854
C02767=1053.191,-0.272,-72.832,170.801,31.152,155.854
C02768=1053.185,-0.522,-72.817,170.799,31.150,155.854
C02769=1053.180,-0.771,-72.802,170.797,31.147,155.853
C02770=1053.174,-1.021,-72.787,170.796,31.145,155.853
C02771=1053.168,-1.270,-72.772,170.794,31.143,155.853
C02772=1053.162,-1.519,-72.757,170.793,31.141,155.853
C02773=1053.155,-1.769,-72.742,170.791,31.139,155.852
C02774=1053.149,-2.018,-72.728,170.789,31.137,155.852
C02775=1053.142,-2.301,-72.711,170.787,31.135,155.852
C02776=1053.135,-2.584,-72.695,170.785,31.133,155.851
C02777=1053.129,-2.866,-72.678,170.784,31.130,155.851
C02778=1053.122,-3.148,-72.661,170.782,31.128,155.851
C02779=1053.116,-3.398,-72.647,170.780,31.126,155.850
C02780=1053.109,-3.648,-72.633,170.778,31.124,155.850
C02781=1053.103,-3.896,-72.618,170.776,31.122,155.850
C02782=1053.097,-4.146,-72.603,170.774,31.120,155.850
C02783=1053.090,-4.396,-72.589,170.773,31.118,155.849
C02784=1053.084,-4.645,-72.575,170.772,31.117,155.849
C02785=1053.078,-4.895,-72.560,170.770,31.114,155.849
C02786=1053.071,-5.144,-72.545,170.768,31.112,155.849
C02787=1053.066,-5.394,-72.531,170.766,31.110,155.848
C02788=1053.059,-5.643,-72.517,170.764,31.109,155.848
C02789=1053.052,-5.893,-72.502,170.763,31.107,155.848
C02790=1053.047,-6.143,-72.488,170.761,31.105,155.848
C02791=1053.040,-6.392,-72.474,170.759,31.103,155.847
C02792=1053.034,-6.641,-72.459,170.758,31.101,155.847
C02793=1053.028,-6.891,-72.445,170.756,31.099,155.847
C02794=1053.021,-7.141,-72.430,170.754,31.097,155.847
C02795=1053.015,-7.389,-72.416,170.752,31.095,155.846
C02796=1053.009,-7.640,-72.402,170.751,31.093,155.846
C02797=1053.003,-7.889,-72.387,170.749,31.091,155.846
C02798=1052.996,-8.139,-72.374,170.747,31.090,155.846
C02799=1052.990,-8.388,-72.359,170.746,31.087,155.845
C02800=1052.984,-8.637,-72.344,170.744,31.085,155.845
C02801=1052.978,-8.887,-72.330,170.742,31.083,155.845
C02802=1052.971,-9.136,-72.316,170.741,31.082,155.845
C02803=1052.965,-9.386,-72.302,170.739,31.080,155.844
C02804=1052.960,-9.635,-72.287,170.737,31.078,155.844
C02805=1052.952,-9.885,-72.273,170.735,31.076,155.844
C02806=1052.947,-10.134,-72.259,170.734,31.074,155.844
C02807=1052.941,-10.384,-72.244,170.732,31.072,155.843
C02808=1052.934,-10.634,-72.230,170.730,31.070,155.843
C02809=1052.928,-10.883,-72.216,170.729,31.068,155.843
C02810=1052.922,-11.133,-72.201,170.727,31.066,155.843
C02811=1052.915,-11.382,-72.187,170.725,31.064,155.842
C02812=1052.909,-11.632,-72.173,170.723,31.063,155.842
C02813=1052.904,-11.881,-72.159,170.722,31.060,155.842
C02814=1052.897,-12.131,-72.144,170.720,31.058,155.842
C02815=1052.891,-12.380,-72.130,170.718,31.057,155.841
C02816=1052.885,-12.630,-72.116,170.717,31.055,155.841
C02817=1052.879,-12.879,-72.102,170.715,31.053,155.841
C02818=1052.872,-13.129,-72.088,170.713,31.051,155.841
C02819=1052.866,-13.378,-72.073,170.711,31.049,155.840
C02820=1052.860,-13.628,-72.059,170.710,31.047,155.840
C02821=1052.854,-13.878,-72.046,170.708,31.045,155.840
C02822=1052.848,-14.127,-72.031,170.706,31.043,155.840
C02823=1052.842,-14.377,-72.018,170.705,31.041,155.839
C02824=1052.836,-14.625,-72.003,170.703,31.040,155.839
C02825=1052.830,-14.876,-71.989,170.701,31.038,155.839
C02826=1052.823,-15.124,-71.975,170.699,31.035,155.839
C02827=1052.817,-15.375,-71.961,170.697,31.034,155.838
C02828=1052.811,-15.624,-71.947,170.696,31.032,155.838
C02829=1052.805,-15.874,-71.932,170.694,31.030,155.838
C02830=1052.798,-16.123,-71.919,170.692,31.028,155.838
C02831=1052.792,-16.373,-71.905,170.691,31.026,155.837
C02832=1052.786,-16.622,-71.891,170.689,31.025,155.837
C02833=1052.780,-16.872,-71.877,170.687,31.022,155.837
C02834=1052.773,-17.121,-71.863,170.685,31.021,155.837
C02835=1052.766,-17.371,-71.849,170.684,31.019,155.837
C02836=1052.761,-17.620,-71.835,170.682,31.017,155.836
C02837=1052.754,-17.870,-71.822,170.680,31.015,155.836
C02838=1052.749,-18.120,-71.808,170.678,31.014,155.836
C02839=1052.741,-18.400,-71.792,170.676,31.012,155.836
C02840=1052.734,-18.681,-71.776,170.674,31.009,155.835
C02841=1052.727,-18.962,-71.760,170.672,31.007,155.835
C02842=1052.720,-19.243,-71.745,170.671,31.005,155.835
C02843=1052.714,-19.493,-71.731,170.669,31.004,155.835
C02844=1052.708,-19.742,-71.717,170.667,31.001,155.834
C02845=1052.701,-19.991,-71.703,170.665,31.000,155.834
C02846=1052.695,-20.241,-71.690,170.663,30.998,155.834
C02847=1052.689,-20.490,-71.676,170.661,30.996,155.834
C02848=1052.682,-20.740,-71.662,170.659,30.994,155.833
C02849=1052.677,-20.990,-71.648,170.659,30.993,155.833
C02850=1052.670,-21.239,-71.634,170.657,30.991,155.833
C02851=1052.664,-21.488,-71.621,170.655,30.989,155.833
C02852=1052.658,-21.738,-71.607,170.653,30.987,155.833
C02853=1052.651,-21.988,-71.593,170.651,30.985,155.832
C02854=1052.646,-22.238,-71.580,170.649,30.983,155.832
C02855=1052.640,-22.487,-71.566,170.647,30.982,155.832
C02856=1052.633,-22.737,-71.553,170.646,30.980,155.832
C02857=1052.627,-22.986,-71.538,170.644,30.978,155.831
C02858=1052.620,-23.236,-71.524,170.642,30.976,155.831
C02859=1052.614,-23.485,-71.511,170.641,30.975,155.831
C02860=1052.609,-23.735,-71.497,170.639,30.972,155.831
C02861=1052.602,-23.985,-71.484,170.637,30.971,155.831
C02862=1052.596,-24.234,-71.470,170.635,30.969,155.830
C02863=1052.590,-24.483,-71.456,170.634,30.967,155.830
C02864=1052.583,-24.733,-71.443,170.632,30.965,155.830
C02865=1052.578,-24.983,-71.429,170.630,30.964,155.830
C02866=1052.572,-25.232,-71.416,170.628,30.961,155.829
C02867=1052.565,-25.481,-71.402,170.626,30.960,155.829
C02868=1052.559,-25.732,-71.388,170.624,30.958,155.829
C02869=1052.553,-25.980,-71.374,170.622,30.956,155.829
C02870=1052.547,-26.230,-71.361,170.622,30.954,155.828
C02871=1052.540,-26.480,-71.347,170.620,30.953,155.828
C02872=1052.534,-26.729,-71.333,170.618,30.951,155.828
C02873=1052.528,-26.978,-71.320,170.616,30.949,155.828
C02874=1052.522,-27.229,-71.307,170.614,30.948,155.828
C02875=1052.516,-27.479,-71.293,170.612,30.945,155.827
C02876=1052.510,-27.728,-71.280,170.610,30.944,155.827
C02877=1052.503,-27.978,-71.267,170.608,30.942,155.827
C02878=1052.497,-28.227,-71.253,170.607,30.940,155.827
C02879=1052.491,-28.476,-71.240,170.605,30.939,155.827
C02880=1052.484,-28.726,-71.227,170.603,30.937,155.826
C02881=1052.478,-28.976,-71.213,170.601,30.935,155.826
C02882=1052.472,-29.225,-71.199,170.599,30.934,155.826
C02883=1052.466,-29.474,-71.186,170.597,30.932,155.826
C02884=1052.459,-29.724,-71.172,170.595,30.930,155.826
C02885=1052.453,-29.974,-71.159,170.595,30.928,155.825
C02886=1052.447,-30.223,-71.146,170.593,30.927,155.825
C02887=1052.441,-30.473,-71.133,170.591,30.925,155.825
C02888=1052.434,-30.723,-71.120,170.589,30.923,155.825
C02889=1052.428,-30.972,-71.106,170.587,30.922,155.825
C02890=1052.421,-31.221,-71.093,170.585,30.920,155.824
C02891=1052.416,-31.471,-71.079,170.583,30.918,155.824
C02892=1052.409,-31.721,-71.066,170.582,30.917,155.824
C02893=1052.403,-31.971,-71.053,170.580,30.915,155.824
C02894=1052.397,-32.220,-71.040,170.578,30.913,155.824
C02895=1052.391,-32.469,-71.026,170.576,30.911,155.823
C02896=1052.384,-32.719,-71.013,170.574,30.910,155.823
C02897=1052.378,-32.968,-71.000,170.572,30.908,155.823
C02898=1052.372,-33.218,-70.987,170.570,30.906,155.823
C02899=1052.366,-33.468,-70.974,170.568,30.905,155.823
C02900=1052.359,-33.717,-70.960,170.567,30.903,155.822
C02901=1052.353,-33.967,-70.947,170.565,30.901,155.822
C02902=1052.347,-34.217,-70.934,170.563,30.899,155.822
C02903=1052.340,-34.497,-70.919,170.561,30.897,155.822
C02904=1052.333,-34.777,-70.904,170.559,30.896,155.822
C02905=1052.326,-35.057,-70.889,170.557,30.894,155.821
C02906=1052.319,-35.337,-70.875,170.555,30.892,155.821
C02907=1052.313,-35.587,-70.861,170.554,30.890,155.821
C02908=1052.307,-35.836,-70.848,170.552,30.888,155.821
C02909=1052.301,-36.086,-70.835,170.550,30.887,155.821
C02910=1052.295,-36.335,-70.822,170.548,30.885,155.820
C02911=1052.288,-36.584,-70.809,170.546,30.883,155.820
C02912=1052.283,-36.834,-70.796,170.544,30.882,155.820
C02913=1052.276,-37.084,-70.783,170.542,30.880,155.820
C02914=1052.270,-37.333,-70.769,170.541,30.879,155.820
C02915=1052.264,-37.583,-70.757,170.539,30.876,155.819
C02916=1052.258,-37.833,-70.743,170.537,30.875,155.819
C02917=1052.252,-38.082,-70.730,170.535,30.873,155.819
C02918=1052.246,-38.332,-70.717,170.533,30.872,155.819
C02919=1052.240,-38.581,-70.704,170.531,30.870,155.819
C02920=1052.234,-38.831,-70.691,170.529,30.868,155.818
C02921=1052.226,-39.081,-70.678,170.528,30.867,155.818
C02922=1052.220,-39.330,-70.665,170.526,30.865,155.818
C02923=1052.214,-39.580,-70.653,170.524,30.863,155.818
C02924=1052.208,-39.829,-70.639,170.522,30.862,155.818
C02925=1052.202,-40.079,-70.627,170.520,30.860,155.818
C02926=1052.196,-40.328,-70.613,170.518,30.859,155.817
C02927=1052.189,-40.578,-70.601,170.516,30.857,155.817
C02928=1052.183,-40.827,-70.588,170.515,30.856,155.817
C02929=1052.176,-41.078,-70.575,170.513,30.854,155.817
C02930=1052.170,-41.327,-70.562,170.511,30.852,155.817
C02931=1052.164,-41.577,-70.549,170.509,30.851,155.816
C02932=1052.157,-41.826,-70.537,170.507,30.849,155.816
C02933=1052.152,-42.076,-70.524,170.505,30.848,155.816
C02934=1052.145,-42.325,-70.511,170.503,30.846,155.816
C02935=1052.139,-42.575,-70.498,170.501,30.844,155.816
C02936=1052.133,-42.824,-70.485,170.500,30.843,155.816
C02937=1052.127,-43.074,-70.473,170.498,30.841,155.815
C02938=1052.120,-43.323,-70.460,170.496,30.840,155.815
C02939=1052.114,-43.573,-70.447,170.494,30.838,155.815
C02940=1052.108,-43.823,-70.435,170.492,30.837,155.815
C02941=1052.102,-44.072,-70.422,170.490,30.835,155.815
C02942=1052.095,-44.322,-70.409,170.488,30.834,155.815
C02943=1052.089,-44.572,-70.396,170.487,30.832,155.815
C02944=1052.083,-44.821,-70.383,170.485,30.830,155.814
C02945=1052.077,-45.071,-70.371,170.483,30.828,155.814
C02946=1052.071,-45.321,-70.358,170.481,30.827,155.814
C02947=1052.064,-45.570,-70.346,170.479,30.825,155.814
C02948=1052.058,-45.819,-70.332,170.477,30.824,155.814
C02949=1052.052,-46.069,-70.320,170.475,30.822,155.813
C02950=1052.046,-46.319,-70.307,170.473,30.821,155.813
C02951=1052.040,-46.568,-70.294,170.472,30.819,155.813
C02952=1052.033,-46.818,-70.282,170.470,30.818,155.813
C02953=1052.027,-47.068,-70.269,170.468,30.816,155.813
C02954=1052.021,-47.317,-70.256,170.466,30.815,155.813
C02955=1052.015,-47.567,-70.244,170.464,30.813,155.812
C02956=1052.009,-47.817,-70.232,170.462,30.812,155.812
C02957=1052.003,-48.067,-70.219,170.460,30.810,155.812
C02958=1051.996,-48.316,-70.206,170.459,30.808,155.812
C02959=1051.991,-48.565,-70.194,170.457,30.807,155.812
C02960=1051.984,-48.815,-70.182,170.455,30.805,155.812
C02961=1051.979,-49.064,-70.169,170.453,30.804,155.811
C02962=1051.972,-49.314,-70.156,170.451,30.802,155.811
C02963=1051.966,-49.564,-70.143,170.449,30.801,155.811
C02964=1051.960,-49.813,-70.131,170.447,30.799,155.811
C02965=1051.954,-50.063,-70.119,170.445,30.798,155.811
C02966=1051.948,-50.312,-70.106,170.444,30.796,155.811
C02967=1051.940,-50.593,-70.092,170.442,30.795,155.810
C02968=1051.933,-50.873,-70.078,170.440,30.793,155.810
C02969=1051.926,-51.154,-70.065,170.437,30.791,155.810
C02970=1051.919,-51.435,-70.050,170.435,30.790,155.810
C02971=1051.913,-51.684,-70.039,170.433,30.788,155.810
C02972=1051.907,-51.934,-70.026,170.431,30.787,155.810
C02973=1051.900,-52.184,-70.014,170.430,30.786,155.810
C02974=1051.894,-52.433,-70.001,170.428,30.784,155.810
C02975=1051.887,-52.682,-69.989,170.426,30.783,155.809
C02976=1051.880,-52.932,-69.977,170.424,30.782,155.809
C02977=1051.875,-53.182,-69.964,170.422,30.780,155.809
C02978=1051.868,-53.431,-69.952,170.420,30.779,155.809
C02979=1051.862,-53.681,-69.940,170.418,30.777,155.809
C02980=1051.855,-53.931,-69.928,170.416,30.776,155.809
C02981=1051.849,-54.181,-69.915,170.414,30.774,155.809
C02982=1051.843,-54.430,-69.903,170.412,30.773,155.808
C02983=1051.836,-54.680,-69.891,170.410,30.771,155.808
C02984=1051.831,-54.929,-69.879,170.408,30.770,155.808
C02985=1051.824,-55.179,-69.867,170.406,30.769,155.808
C02986=1051.818,-55.429,-69.855,170.404,30.767,155.808
C02987=1051.812,-55.678,-69.843,170.402,30.766,155.808
C02988=1051.805,-55.928,-69.831,170.400,30.765,155.808
C02989=1051.799,-56.178,-69.818,170.399,30.763,155.808
C02990=1051.792,-56.427,-69.806,170.397,30.762,155.807
C02991=1051.786,-56.677,-69.794,170.395,30.761,155.807
C02992=1051.780,-56.927,-69.782,170.393,30.759,155.807
C02993=1051.773,-57.176,-69.770,170.391,30.758,155.807
C02994=1051.768,-57.425,-69.758,170.389,30.756,155.807
C02995=1051.761,-57.675,-69.746,170.387,30.755,155.807
C02996=1051.755,-57.924,-69.734,170.385,30.754,155.807
C02997=1051.749,-58.174,-69.721,170.384,30.752,155.806
C02998=1051.742,-58.424,-69.709,170.381,30.751,155.806
C02999=1051.735,-58.673,-69.697,170.379,30.750,155.806
C03000=1051.730,-58.923,-69.685,170.377,30.748,155.806
C03001=1051.724,-59.172,-69.673,170.375,30.747,155.806
C03002=1051.718,-59.423,-69.661,170.373,30.746,155.806
C03003=1051.711,-59.672,-69.649,170.371,30.744,155.806
C03004=1051.705,-59.922,-69.637,170.369,30.743,155.806
C03005=1051.699,-60.172,-69.625,170.368,30.742,155.806
C03006=1051.693,-60.421,-69.613,170.366,30.740,155.805
C03007=1051.686,-60.670,-69.601,170.364,30.739,155.805
C03008=1051.680,-60.920,-69.589,170.362,30.738,155.805
C03009=1051.674,-61.170,-69.577,170.360,30.736,155.805
C03010=1051.667,-61.420,-69.565,170.358,30.735,155.805
C03011=1051.662,-61.669,-69.553,170.356,30.733,155.805
C03012=1051.655,-61.919,-69.541,170.354,30.732,155.805
C03013=1051.649,-62.168,-69.529,170.352,30.731,155.805
C03014=1051.643,-62.418,-69.517,170.350,30.729,155.804
C03015=1051.637,-62.668,-69.506,170.348,30.728,155.804
C03016=1051.630,-62.917,-69.494,170.346,30.727,155.804
C03017=1051.624,-63.167,-69.481,170.344,30.725,155.804
C03018=1051.618,-63.417,-69.469,170.342,30.724,155.804
C03019=1051.612,-63.666,-69.458,170.340,30.723,155.804
C03020=1051.606,-63.916,-69.446,170.339,30.721,155.804
C03021=1051.599,-64.166,-69.434,170.337,30.720,155.804
C03022=1051.593,-64.415,-69.422,170.335,30.719,155.804
C03023=1051.587,-64.665,-69.411,170.333,30.718,155.803
C03024=1051.581,-64.914,-69.399,170.331,30.716,155.803
C03025=1051.574,-65.164,-69.387,170.329,30.715,155.803
C03026=1051.569,-65.414,-69.376,170.326,30.714,155.803
C03027=1051.563,-65.663,-69.363,170.324,30.712,155.803
C03028=1051.556,-65.913,-69.351,170.322,30.711,155.803
C03029=1051.550,-66.162,-69.340,170.321,30.710,155.803
C03030=1051.544,-66.412,-69.328,170.319,30.709,155.803
C03031=1051.537,-66.694,-69.315,170.317,30.707,155.803
C03032=1051.530,-66.975,-69.301,170.314,30.705,155.802
C03033=1051.523,-67.257,-69.288,170.312,30.704,155.802
C03034=1051.516,-67.540,-69.275,170.310,30.702,155.802
C03035=1051.510,-67.789,-69.263,170.308,30.701,155.802
C03036=1051.504,-68.039,-69.251,170.307,30.700,155.802
C03037=1051.498,-68.288,-69.240,170.305,30.699,155.802
C03038=1051.492,-68.538,-69.228,170.302,30.697,155.802
C03039=1051.486,-68.788,-69.216,170.300,30.696,155.802
C03040=1051.480,-69.037,-69.205,170.298,30.695,155.802
C03041=1051.473,-69.287,-69.194,170.296,30.694,155.801
C03042=1051.467,-69.537,-69.181,170.294,30.692,155.801
C03043=1051.461,-69.786,-69.169,170.292,30.691,155.801
C03044=1051.455,-70.036,-69.158,170.291,30.690,155.801
C03045=1051.449,-70.285,-69.147,170.289,30.689,155.801
C03046=1051.443,-70.536,-69.135,170.287,30.687,155.801
C03047=1051.437,-70.785,-69.123,170.285,30.686,155.801
C03048=1051.431,-71.035,-69.112,170.283,30.685,155.801
C03049=1051.424,-71.284,-69.100,170.280,30.684,155.801
C03050=1051.419,-71.534,-69.088,170.278,30.682,155.801
C03051=1051.413,-71.784,-69.076,170.276,30.681,155.800
C03052=1051.407,-72.033,-69.066,170.275,30.680,155.800
C03053=1051.400,-72.283,-69.054,170.273,30.679,155.800
C03054=1051.395,-72.533,-69.042,170.271,30.677,155.800
C03055=1051.389,-72.782,-69.030,170.269,30.676,155.800
C03056=1051.382,-73.032,-69.019,170.267,30.675,155.800
C03057=1051.376,-73.281,-69.007,170.265,30.674,155.800
C03058=1051.370,-73.531,-68.996,170.263,30.672,155.800
C03059=1051.365,-73.781,-68.985,170.260,30.671,155.800
C03060=1051.358,-74.031,-68.973,170.259,30.669,155.800
C03061=1051.353,-74.280,-68.962,170.257,30.669,155.799
C03062=1051.346,-74.530,-68.950,170.255,30.668,155.799
C03063=1051.340,-74.780,-68.939,170.253,30.666,155.799
C03064=1051.334,-75.029,-68.928,170.251,30.665,155.799
C03065=1051.327,-75.279,-68.916,170.249,30.664,155.799
C03066=1051.322,-75.528,-68.905,170.247,30.663,155.799
C03067=1051.315,-75.779,-68.894,170.244,30.662,155.799
C03068=1051.309,-76.027,-68.882,170.242,30.661,155.799
C03069=1051.303,-76.278,-68.871,170.241,30.660,155.799
C03070=1051.297,-76.527,-68.860,170.239,30.658,155.799
C03071=1051.290,-76.777,-68.848,170.237,30.657,155.799
C03072=1051.284,-77.027,-68.837,170.235,30.656,155.799
C03073=1051.278,-77.276,-68.826,170.233,30.655,155.799
C03074=1051.272,-77.526,-68.814,170.231,30.654,155.798
C03075=1051.266,-77.775,-68.803,170.229,30.653,155.798
C03076=1051.260,-78.026,-68.792,170.226,30.652,155.798
C03077=1051.253,-78.275,-68.782,170.224,30.651,155.798
C03078=1051.246,-78.524,-68.770,170.223,30.649,155.798
C03079=1051.241,-78.774,-68.759,170.221,30.648,155.798
C03080=1051.234,-79.024,-68.747,170.219,30.647,155.798
C03081=1051.229,-79.274,-68.737,170.217,30.646,155.798
C03082=1051.222,-79.523,-68.725,170.215,30.645,155.798
C03083=1051.216,-79.773,-68.714,170.212,30.644,155.798
C03084=1051.210,-80.023,-68.702,170.210,30.643,155.798
C03085=1051.204,-80.272,-68.692,170.208,30.642,155.798
C03086=1051.197,-80.522,-68.681,170.206,30.641,155.798
C03087=1051.191,-80.772,-68.670,170.205,30.640,155.798
C03088=1051.185,-81.021,-68.658,170.203,30.639,155.798
C03089=1051.179,-81.271,-68.647,170.201,30.638,155.798
C03090=1051.172,-81.521,-68.637,170.198,30.637,155.798
C03091=1051.166,-81.770,-68.626,170.196,30.636,155.798
C03092=1051.160,-82.020,-68.614,170.194,30.635,155.797
C03093=1051.154,-82.270,-68.604,170.192,30.634,155.797
C03094=1051.147,-82.520,-68.593,170.190,30.633,155.797
C03095=1051.140,-82.804,-68.580,170.188,30.632,155.797
C03096=1051.134,-83.087,-68.568,170.186,30.631,155.797
C03097=1051.126,-83.371,-68.555,170.183,30.629,155.797
C03098=1051.119,-83.655,-68.543,170.181,30.629,155.797
C03099=1051.112,-83.905,-68.532,170.179,30.628,155.797
C03100=1051.107,-84.154,-68.521,170.177,30.627,155.797
C03101=1051.100,-84.405,-68.510,170.175,30.626,155.797
C03102=1051.094,-84.654,-68.500,170.172,30.625,155.797
C03103=1051.087,-84.904,-68.488,170.170,30.624,155.797
C03104=1051.082,-85.153,-68.478,170.168,30.623,155.797
C03105=1051.075,-85.403,-68.467,170.167,30.622,155.797
C03106=1051.069,-85.653,-68.456,170.165,30.621,155.797
C03107=1051.063,-85.902,-68.445,170.163,30.620,155.797
C03108=1051.056,-86.152,-68.434,170.160,30.619,155.797
C03109=1051.050,-86.402,-68.424,170.158,30.618,155.797
C03110=1051.045,-86.651,-68.413,170.156,30.617,155.797
C03111=1051.038,-86.901,-68.402,170.154,30.616,155.797
C03112=1051.032,-87.151,-68.391,170.152,30.615,155.797
C03113=1051.025,-87.401,-68.380,170.150,30.614,155.797
C03114=1051.019,-87.650,-68.370,170.149,30.613,155.796
C03115=1051.013,-87.899,-68.359,170.146,30.612,155.796
C03116=1051.007,-88.150,-68.348,170.144,30.611,155.796
C03117=1051.000,-88.399,-68.337,170.142,30.610,155.796
C03118=1050.995,-88.649,-68.327,170.140,30.609,155.796
C03119=1050.989,-88.899,-68.316,170.138,30.609,155.796
C03120=1050.982,-89.148,-68.306,170.136,30.608,155.796
C03121=1050.976,-89.398,-68.295,170.133,30.607,155.796
C03122=1050.970,-89.648,-68.283,170.131,30.606,155.796
C03123=1050.964,-89.897,-68.273,170.129,30.605,155.796
C03124=1050.958,-90.147,-68.262,170.128,30.604,155.796
C03125=1050.952,-90.397,-68.251,170.126,30.603,155.796
C03126=1050.945,-90.647,-68.242,170.124,30.602,155.796
C03127=1050.940,-90.896,-68.231,170.121,30.601,155.796
C03128=1050.933,-91.146,-68.219,170.119,30.600,155.796
C03129=1050.927,-91.395,-68.209,170.117,30.600,155.796
C03130=1050.921,-91.645,-68.198,170.115,30.599,155.796
C03131=1050.915,-91.895,-68.189,170.113,30.598,155.796
C03132=1050.909,-92.145,-68.177,170.111,30.597,155.796
C03133=1050.903,-92.394,-68.167,170.109,30.596,155.796
C03134=1050.896,-92.644,-68.156,170.107,30.595,155.796
C03135=1050.891,-92.893,-68.145,170.105,30.594,155.796
C03136=1050.885,-93.144,-68.135,170.103,30.594,155.796
C03137=1050.878,-93.393,-68.125,170.101,30.593,155.796
C03138=1050.872,-93.643,-68.114,170.099,30.592,155.796
C03139=1050.866,-93.892,-68.103,170.096,30.591,155.796
C03140=1050.860,-94.143,-68.093,170.094,30.590,155.796
C03141=1050.854,-94.392,-68.082,170.092,30.589,155.796
C03142=1050.848,-94.641,-68.072,170.090,30.588,155.796
C03143=1050.842,-94.891,-68.062,170.089,30.587,155.796
C03144=1050.835,-95.141,-68.051,170.087,30.587,155.796
C03145=1050.829,-95.391,-68.040,170.084,30.585,155.796
C03146=1050.824,-95.640,-68.029,170.082,30.584,155.796
C03147=1050.817,-95.890,-68.020,170.080,30.584,155.796
C03148=1050.812,-96.139,-68.009,170.078,30.583,155.796
C03149=1050.805,-96.389,-67.998,170.076,30.582,155.796
C03150=1050.799,-96.639,-67.988,170.073,30.581,155.796
C03151=1050.793,-96.889,-67.977,170.071,30.580,155.796
C03152=1050.787,-97.139,-67.967,170.069,30.580,155.796
C03153=1050.782,-97.388,-67.957,170.068,30.579,155.796
C03154=1050.774,-97.638,-67.946,170.066,30.578,155.796
C03155=1050.768,-97.888,-67.936,170.064,30.578,155.796
C03156=1050.763,-98.137,-67.925,170.061,30.577,155.796
C03157=1050.756,-98.387,-67.916,170.059,30.576,155.796
C03158=1050.751,-98.637,-67.905,170.057,30.575,155.796
C03159=1050.743,-98.923,-67.893,170.054,30.574,155.796
C03160=1050.736,-99.209,-67.881,170.052,30.573,155.796
C03161=1050.729,-99.495,-67.870,170.049,30.573,155.796
C03162=1050.721,-99.782,-67.858,170.047,30.572,155.796
C03163=1050.715,-100.032,-67.848,170.046,30.571,155.796
C03164=1050.709,-100.281,-67.838,170.043,30.570,155.796
C03165=1050.703,-100.531,-67.828,170.041,30.569,155.796
C03166=1050.697,-100.780,-67.818,170.039,30.569,155.796
C03167=1050.691,-101.030,-67.808,170.037,30.568,155.796
C03168=1050.684,-101.280,-67.797,170.035,30.568,155.796
C03169=1050.678,-101.530,-67.787,170.033,30.567,155.796
C03170=1050.672,-101.780,-67.776,170.030,30.566,155.796
C03171=1050.666,-102.029,-67.767,170.028,30.565,155.796
C03172=1050.660,-102.279,-67.757,170.026,30.565,155.796
C03173=1050.654,-102.529,-67.746,170.024,30.564,155.796
C03174=1050.648,-102.778,-67.737,170.023,30.563,155.796
C03175=1050.641,-103.028,-67.726,170.020,30.563,155.796
C03176=1050.636,-103.278,-67.716,170.018,30.562,155.796
C03177=1050.629,-103.528,-67.706,170.016,30.562,155.796
C03178=1050.623,-103.777,-67.696,170.014,30.561,155.796
C03179=1050.618,-104.028,-67.686,170.011,30.560,155.796
C03180=1050.611,-104.277,-67.676,170.009,30.559,155.796
C03181=1050.605,-104.527,-67.666,170.007,30.559,155.796
C03182=1050.598,-104.776,-67.656,170.005,30.558,155.796
C03183=1050.593,-105.026,-67.646,170.003,30.558,155.796
C03184=1050.587,-105.276,-67.636,170.000,30.557,155.796
C03185=1050.580,-105.525,-67.626,169.998,30.556,155.796
C03186=1050.574,-105.776,-67.615,169.997,30.556,155.796
C03187=1050.568,-106.025,-67.606,169.995,30.555,155.796
C03188=1050.562,-106.275,-67.595,169.993,30.555,155.796
C03189=1050.556,-106.524,-67.586,169.990,30.553,155.796
C03190=1050.549,-106.774,-67.576,169.988,30.553,155.796
C03191=1050.544,-107.024,-67.566,169.986,30.553,155.796
C03192=1050.537,-107.273,-67.556,169.984,30.552,155.796
C03193=1050.531,-107.523,-67.546,169.982,30.551,155.796
C03194=1050.525,-107.773,-67.537,169.979,30.551,155.796
C03195=1050.519,-108.023,-67.527,169.977,30.550,155.796
C03196=1050.513,-108.272,-67.516,169.975,30.550,155.796
C03197=1050.507,-108.522,-67.507,169.973,30.549,155.796
C03198=1050.501,-108.772,-67.497,169.972,30.548,155.796
C03199=1050.495,-109.022,-67.488,169.969,30.548,155.796
C03200=1050.488,-109.271,-67.477,169.967,30.548,155.797
C03201=1050.482,-109.521,-67.468,169.965,30.547,155.797
C03202=1050.476,-109.771,-67.458,169.963,30.546,155.797
C03203=1050.470,-110.020,-67.449,169.960,30.546,155.797
C03204=1050.463,-110.270,-67.439,169.958,30.546,155.797
C03205=1050.458,-110.520,-67.428,169.956,30.545,155.797
C03206=1050.452,-110.769,-67.419,169.954,30.544,155.797
C03207=1050.445,-111.019,-67.409,169.952,30.544,155.797
C03208=1050.439,-111.269,-67.400,169.949,30.543,155.797
C03209=1050.433,-111.519,-67.390,169.947,30.543,155.797
C03210=1050.427,-111.769,-67.380,169.946,30.542,155.797
C03211=1050.421,-112.018,-67.371,169.944,30.542,155.797
C03212=1050.415,-112.268,-67.361,169.941,30.541,155.797
C03213=1050.408,-112.517,-67.351,169.939,30.540,155.797
C03214=1050.402,-112.767,-67.341,169.937,30.540,155.797
C03215=1050.396,-113.017,-67.332,169.935,30.540,155.797
C03216=1050.390,-113.267,-67.322,169.933,30.539,155.797
C03217=1050.384,-113.517,-67.312,169.930,30.539,155.797
C03218=1050.378,-113.767,-67.303,169.928,30.538,155.797
C03219=1050.372,-114.016,-67.293,169.926,30.538,155.797
C03220=1050.366,-114.266,-67.283,169.924,30.537,155.797
C03221=1050.359,-114.516,-67.274,169.921,30.537,155.798
C03222=1050.353,-114.766,-67.264,169.919,30.537,155.798
C03223=1050.346,-115.051,-67.254,169.918,30.536,155.798
C03224=1050.339,-115.336,-67.243,169.915,30.536,155.798
C03225=1050.333,-115.621,-67.232,169.913,30.535,155.798
C03226=1050.325,-115.906,-67.221,169.910,30.534,155.798
C03227=1050.319,-116.156,-67.212,169.908,30.534,155.798
C03228=1050.313,-116.406,-67.202,169.906,30.534,155.798
C03229=1050.307,-116.655,-67.192,169.903,30.533,155.798
C03230=1050.301,-116.905,-67.183,169.901,30.533,155.798
C03231=1050.295,-117.155,-67.173,169.899,30.533,155.798
C03232=1050.289,-117.404,-67.164,169.897,30.532,155.798
C03233=1050.283,-117.654,-67.155,169.894,30.532,155.798
C03234=1050.277,-117.904,-67.145,169.892,30.531,155.798
C03235=1050.270,-118.153,-67.136,169.890,30.531,155.799
C03236=1050.264,-118.403,-67.126,169.888,30.531,155.799
C03237=1050.257,-118.653,-67.117,169.886,30.530,155.799
C03238=1050.251,-118.903,-67.107,169.884,30.530,155.799
C03239=1050.245,-119.153,-67.098,169.882,30.530,155.799
C03240=1050.240,-119.402,-67.089,169.880,30.529,155.799
C03241=1050.234,-119.652,-67.080,169.877,30.529,155.799
C03242=1050.227,-119.902,-67.070,169.875,30.528,155.799
C03243=1050.221,-120.151,-67.061,169.873,30.528,155.799
C03244=1050.214,-120.401,-67.052,169.871,30.528,155.799
C03245=1050.208,-120.651,-67.042,169.869,30.527,155.799
C03246=1050.202,-120.901,-67.033,169.866,30.527,155.799
C03247=1050.197,-121.150,-67.024,169.864,30.527,155.799
C03248=1050.191,-121.400,-67.014,169.862,30.526,155.800
C03249=1050.184,-121.650,-67.005,169.860,30.526,155.800
C03250=1050.178,-121.900,-66.995,169.857,30.526,155.800
C03251=1050.172,-122.150,-66.987,169.856,30.525,155.800
C03252=1050.166,-122.399,-66.978,169.854,30.525,155.800
C03253=1050.160,-122.649,-66.968,169.852,30.525,155.800
C03254=1050.154,-122.898,-66.959,169.849,30.525,155.800
C03255=1050.148,-123.149,-66.950,169.847,30.524,155.800
C03256=1050.142,-123.399,-66.940,169.845,30.524,155.800
C03257=1050.135,-123.647,-66.932,169.843,30.524,155.800
C03258=1050.129,-123.897,-66.922,169.840,30.523,155.800
C03259=1050.123,-124.148,-66.913,169.838,30.523,155.800
C03260=1050.117,-124.397,-66.904,169.836,30.523,155.801
C03261=1050.111,-124.647,-66.894,169.834,30.523,155.801
C03262=1050.105,-124.897,-66.886,169.831,30.522,155.801
C03263=1050.099,-125.146,-66.877,169.829,30.522,155.801
C03264=1050.093,-125.396,-66.867,169.827,30.522,155.801
C03265=1050.086,-125.646,-66.859,169.825,30.522,155.801
C03266=1050.080,-125.895,-66.850,169.822,30.522,155.801
C03267=1050.074,-126.145,-66.840,169.821,30.521,155.801
C03268=1050.068,-126.396,-66.831,169.819,30.521,155.801
C03269=1050.061,-126.645,-66.822,169.817,30.521,155.802
C03270=1050.056,-126.894,-66.813,169.814,30.521,155.802
C03271=1050.050,-127.145,-66.804,169.812,30.520,155.802
C03272=1050.043,-127.394,-66.795,169.810,30.520,155.802
C03273=1050.038,-127.643,-66.786,169.808,30.520,155.802
C03274=1050.032,-127.894,-66.777,169.805,30.520,155.802
C03275=1050.027,-128.143,-66.767,169.803,30.519,155.802
C03276=1050.023,-128.393,-66.757,169.801,30.518,155.802
C03277=1050.020,-128.643,-66.745,169.799,30.516,155.802
C03278=1050.018,-128.893,-66.734,169.798,30.514,155.801
C03279=1050.017,-129.144,-66.721,169.797,30.512,155.801
C03280=1050.018,-129.394,-66.709,169.795,30.508,155.801
C03281=1050.019,-129.645,-66.695,169.793,30.504,155.800
C03282=1050.022,-129.894,-66.682,169.793,30.500,155.799
C03283=1050.025,-130.145,-66.667,169.792,30.496,155.799
C03284=1050.030,-130.396,-66.650,169.790,30.490,155.798
C03285=1050.035,-130.647,-66.634,169.790,30.485,155.797
C03286=1050.041,-130.896,-66.618,169.789,30.479,155.796
C03287=1049.677,-130.920,-66.844,169.743,30.648,155.828
C03288=1049.671,-130.671,-66.860,169.744,30.654,155.829
C03289=1049.666,-130.420,-66.877,169.745,30.660,155.830
C03290=1049.661,-130.169,-66.892,169.746,30.665,155.831
C03291=1049.658,-129.918,-66.907,169.747,30.670,155.832
C03292=1049.656,-129.668,-66.922,169.748,30.674,155.832
C03293=1049.654,-129.418,-66.935,169.749,30.677,155.833
C03294=1049.654,-129.167,-66.948,169.751,30.681,155.833
C03295=1049.654,-128.917,-66.961,169.753,30.683,155.834
C03296=1049.656,-128.667,-66.972,169.753,30.685,155.834
C03297=1049.659,-128.417,-66.983,169.755,30.687,155.834
C03298=1049.662,-128.167,-66.994,169.757,30.689,155.834
C03299=1049.667,-127.917,-67.003,169.759,30.689,155.834
C03300=1049.673,-127.667,-67.013,169.762,30.689,155.834
C03301=1049.679,-127.418,-67.022,169.764,30.690,155.834
C03302=1049.685,-127.168,-67.030,169.766,30.690,155.834
C03303=1049.691,-126.918,-67.040,169.768,30.690,155.834
C03304=1049.697,-126.669,-67.049,169.771,30.690,155.834
C03305=1049.704,-126.419,-67.057,169.773,30.690,155.834
C03306=1049.710,-126.169,-67.067,169.775,30.691,155.833
C03307=1049.716,-125.919,-67.077,169.778,30.691,155.833
C03308=1049.722,-125.670,-67.084,169.780,30.691,155.833
C03309=1049.728,-125.420,-67.094,169.781,30.691,155.833
C03310=1049.734,-125.170,-67.104,169.783,30.692,155.833
C03311=1049.741,-124.920,-67.112,169.786,30.692,155.833
C03312=1049.746,-124.671,-67.121,169.788,30.692,155.833
C03313=1049.753,-124.421,-67.131,169.790,30.692,155.833
C03314=1049.758,-124.171,-67.139,169.792,30.692,155.833
C03315=1049.765,-123.921,-67.149,169.795,30.693,155.833
C03316=1049.772,-123.671,-67.158,169.797,30.693,155.832
C03317=1049.777,-123.422,-67.167,169.799,30.693,155.832
C03318=1049.783,-123.172,-67.176,169.801,30.693,155.832
C03319=1049.789,-122.922,-67.186,169.804,30.694,155.832
C03320=1049.795,-122.672,-67.195,169.806,30.694,155.832
C03321=1049.802,-122.423,-67.204,169.808,30.694,155.832
C03322=1049.807,-122.173,-67.213,169.810,30.695,155.832
C03323=1049.814,-121.923,-67.222,169.813,30.695,155.832
C03324=1049.820,-121.673,-67.232,169.815,30.695,155.832
C03325=1049.826,-121.424,-67.241,169.817,30.695,155.832
C03326=1049.832,-121.173,-67.250,169.818,30.695,155.832
C03327=1049.837,-120.924,-67.259,169.821,30.696,155.831
C03328=1049.844,-120.675,-67.268,169.823,30.696,155.831
C03329=1049.851,-120.425,-67.278,169.825,30.697,155.831
C03330=1049.857,-120.175,-67.287,169.827,30.697,155.831
C03331=1049.863,-119.925,-67.297,169.830,30.697,155.831
C03332=1049.869,-119.675,-67.306,169.832,30.698,155.831
C03333=1049.874,-119.426,-67.315,169.834,30.698,155.831
C03334=1049.880,-119.176,-67.325,169.836,30.698,155.831
C03335=1049.887,-118.926,-67.334,169.839,30.699,155.831
C03336=1049.893,-118.676,-67.344,169.841,30.699,155.831
C03337=1049.900,-118.427,-67.353,169.843,30.699,155.831
C03338=1049.906,-118.177,-67.362,169.845,30.700,155.831
C03339=1049.912,-117.927,-67.372,169.848,30.700,155.831
C03340=1049.918,-117.678,-67.381,169.849,30.700,155.830
C03341=1049.924,-117.427,-67.390,169.851,30.701,155.830
C03342=1049.930,-117.178,-67.400,169.853,30.701,155.830
C03343=1049.936,-116.928,-67.409,169.856,30.702,155.830
C03344=1049.942,-116.678,-67.419,169.858,30.702,155.830
C03345=1049.948,-116.429,-67.428,169.860,30.702,155.830
C03346=1049.954,-116.179,-67.438,169.862,30.703,155.830
C03347=1049.961,-115.929,-67.447,169.865,30.703,155.830
C03348=1049.968,-115.644,-67.458,169.867,30.703,155.830
C03349=1049.975,-115.359,-67.469,169.870,30.704,155.830
C03350=1049.981,-115.074,-67.480,169.872,30.704,155.830
C03351=1049.988,-114.789,-67.490,169.875,30.705,155.830
C03352=1049.995,-114.539,-67.500,169.877,30.706,155.830
C03353=1050.001,-114.289,-67.510,169.879,30.706,155.830
C03354=1050.007,-114.039,-67.519,169.881,30.706,155.830
C03355=1050.013,-113.790,-67.529,169.883,30.707,155.829
C03356=1050.020,-113.541,-67.539,169.885,30.707,155.829
C03357=1050.026,-113.291,-67.549,169.887,30.707,155.829
C03358=1050.032,-113.041,-67.558,169.889,30.708,155.829
C03359=1050.038,-112.791,-67.568,169.892,30.709,155.829
C03360=1050.044,-112.541,-67.577,169.894,30.709,155.829
C03361=1050.050,-112.291,-67.587,169.896,30.709,155.829
C03362=1050.056,-112.041,-67.597,169.898,30.710,155.829
C03363=1050.062,-111.792,-67.607,169.901,30.711,155.829
C03364=1050.068,-111.542,-67.616,169.903,30.711,155.829
C03365=1050.074,-111.292,-67.626,169.905,30.711,155.829
C03366=1050.081,-111.043,-67.636,169.907,30.712,155.829
C03367=1050.087,-110.793,-67.646,169.909,30.713,155.829
C03368=1050.093,-110.543,-67.655,169.911,30.713,155.829
C03369=1050.099,-110.293,-67.665,169.913,30.713,155.829
C03370=1050.106,-110.044,-67.674,169.915,30.714,155.829
C03371=1050.111,-109.794,-67.684,169.917,30.715,155.829
C03372=1050.117,-109.544,-67.695,169.920,30.715,155.829
C03373=1050.124,-109.295,-67.704,169.922,30.715,155.829
C03374=1050.130,-109.045,-67.714,169.924,30.716,155.828
C03375=1050.136,-108.795,-67.723,169.926,30.717,155.829
C03376=1050.142,-108.545,-67.733,169.928,30.717,155.828
C03377=1050.149,-108.296,-67.743,169.931,30.717,155.828
C03378=1050.155,-108.046,-67.753,169.933,30.718,155.828
C03379=1050.161,-107.796,-67.762,169.935,30.719,155.828
C03380=1050.166,-107.546,-67.773,169.937,30.719,155.828
C03381=1050.173,-107.297,-67.783,169.939,30.720,155.828
C03382=1050.179,-107.047,-67.792,169.941,30.720,155.828
C03383=1050.185,-106.798,-67.802,169.943,30.721,155.828
C03384=1050.191,-106.548,-67.813,169.945,30.721,155.828
C03385=1050.197,-106.298,-67.822,169.947,30.722,155.828
C03386=1050.203,-106.048,-67.832,169.950,30.722,155.828
C03387=1050.210,-105.798,-67.842,169.952,30.723,155.828
C03388=1050.217,-105.549,-67.852,169.954,30.724,155.828
C03389=1050.222,-105.299,-67.862,169.956,30.725,155.828
C03390=1050.228,-105.049,-67.872,169.959,30.725,155.828
C03391=1050.235,-104.800,-67.882,169.961,30.725,155.828
C03392=1050.240,-104.550,-67.892,169.963,30.726,155.828
C03393=1050.247,-104.300,-67.903,169.964,30.727,155.828
C03394=1050.253,-104.051,-67.912,169.966,30.728,155.828
C03395=1050.259,-103.801,-67.922,169.969,30.728,155.828
C03396=1050.265,-103.551,-67.933,169.971,30.729,155.828
C03397=1050.271,-103.301,-67.942,169.973,30.729,155.828
C03398=1050.278,-103.052,-67.953,169.975,30.730,155.828
C03399=1050.283,-102.801,-67.963,169.977,30.731,155.828
C03400=1050.289,-102.552,-67.973,169.980,30.732,155.828
C03401=1050.296,-102.303,-67.983,169.982,30.732,155.828
C03402=1050.301,-102.052,-67.993,169.984,30.733,155.828
C03403=1050.308,-101.803,-68.003,169.986,30.733,155.828
C03404=1050.314,-101.553,-68.013,169.988,30.734,155.828
C03405=1050.320,-101.304,-68.024,169.990,30.735,155.828
C03406=1050.327,-101.053,-68.034,169.992,30.736,155.828
C03407=1050.333,-100.804,-68.044,169.994,30.736,155.828
C03408=1050.338,-100.554,-68.054,169.996,30.737,155.828
C03409=1050.345,-100.305,-68.064,169.999,30.737,155.828
C03410=1050.351,-100.055,-68.074,170.001,30.738,155.828
C03411=1050.357,-99.806,-68.085,170.003,30.739,155.828
C03412=1050.364,-99.518,-68.096,170.005,30.740,155.828
C03413=1050.371,-99.232,-68.108,170.008,30.741,155.828
C03414=1050.378,-98.946,-68.119,170.010,30.741,155.828
C03415=1050.386,-98.660,-68.131,170.013,30.742,155.828
C03416=1050.392,-98.410,-68.142,170.014,30.743,155.828
C03417=1050.398,-98.160,-68.152,170.016,30.743,155.828
C03418=1050.404,-97.911,-68.162,170.019,30.744,155.828
C03419=1050.411,-97.661,-68.173,170.021,30.745,155.828
C03420=1050.417,-97.411,-68.183,170.023,30.746,155.828
C03421=1050.422,-97.162,-68.194,170.025,30.747,155.828
C03422=1050.429,-96.912,-68.203,170.027,30.748,155.828
C03423=1050.434,-96.662,-68.214,170.030,30.748,155.828
C03424=1050.441,-96.413,-68.225,170.032,30.749,155.828
C03425=1050.447,-96.162,-68.235,170.034,30.750,155.828
C03426=1050.453,-95.913,-68.246,170.036,30.751,155.828
C03427=1050.459,-95.664,-68.256,170.037,30.751,155.828
C03428=1050.465,-95.414,-68.266,170.039,30.752,155.828
C03429=1050.472,-95.164,-68.277,170.042,30.753,155.828
C03430=1050.477,-94.914,-68.288,170.044,30.754,155.828
C03431=1050.483,-94.664,-68.298,170.046,30.754,155.828
C03432=1050.489,-94.415,-68.308,170.048,30.755,155.828
C03433=1050.495,-94.166,-68.319,170.050,30.756,155.828
C03434=1050.502,-93.916,-68.330,170.053,30.757,155.828
C03435=1050.508,-93.666,-68.340,170.055,30.758,155.828
C03436=1050.513,-93.416,-68.351,170.057,30.759,155.828
C03437=1050.520,-93.167,-68.361,170.058,30.760,155.828
C03438=1050.526,-92.917,-68.372,170.060,30.760,155.828
C03439=1050.532,-92.667,-68.382,170.062,30.761,155.828
C03440=1050.538,-92.417,-68.393,170.065,30.763,155.828
C03441=1050.544,-92.168,-68.404,170.067,30.763,155.828
C03442=1050.551,-91.918,-68.414,170.069,30.764,155.828
C03443=1050.557,-91.669,-68.425,170.071,30.765,155.828
C03444=1050.562,-91.418,-68.435,170.073,30.766,155.828
C03445=1050.569,-91.169,-68.446,170.075,30.767,155.828
C03446=1050.575,-90.919,-68.457,170.078,30.768,155.828
C03447=1050.581,-90.670,-68.467,170.079,30.769,155.828
C03448=1050.587,-90.420,-68.478,170.081,30.770,155.828
C03449=1050.593,-90.170,-68.489,170.083,30.770,155.828
C03450=1050.600,-89.920,-68.499,170.085,30.771,155.828
C03451=1050.605,-89.671,-68.510,170.088,30.772,155.828
C03452=1050.612,-89.421,-68.521,170.090,30.773,155.828
C03453=1050.618,-89.172,-68.531,170.092,30.774,155.828
C03454=1050.624,-88.922,-68.542,170.094,30.775,155.828
C03455=1050.630,-88.672,-68.553,170.096,30.776,155.828
C03456=1050.637,-88.423,-68.564,170.098,30.777,155.828
C03457=1050.642,-88.173,-68.574,170.100,30.778,155.828
C03458=1050.648,-87.922,-68.585,170.102,30.779,155.828
C03459=1050.655,-87.673,-68.595,170.104,30.779,155.829
C03460=1050.661,-87.423,-68.607,170.106,30.780,155.829
C03461=1050.667,-87.174,-68.617,170.108,30.781,155.828
C03462=1050.673,-86.924,-68.628,170.110,30.782,155.829
C03463=1050.680,-86.674,-68.639,170.113,30.783,155.829
C03464=1050.686,-86.425,-68.650,170.115,30.784,155.829
C03465=1050.693,-86.175,-68.660,170.117,30.785,155.829
C03466=1050.698,-85.925,-68.671,170.119,30.786,155.829
C03467=1050.704,-85.676,-68.682,170.121,30.786,155.829
C03468=1050.711,-85.426,-68.693,170.122,30.787,155.829
C03469=1050.717,-85.176,-68.704,170.124,30.788,155.829
C03470=1050.723,-84.926,-68.715,170.127,30.789,155.829
C03471=1050.730,-84.677,-68.725,170.129,30.790,155.829
C03472=1050.735,-84.428,-68.736,170.131,30.791,155.829
C03473=1050.742,-84.177,-68.747,170.133,30.792,155.829
C03474=1050.748,-83.928,-68.758,170.135,30.793,155.829
C03475=1050.755,-83.678,-68.769,170.137,30.794,155.829
C03476=1050.762,-83.394,-68.782,170.140,30.795,155.829
C03477=1050.769,-83.110,-68.794,170.142,30.796,155.829
C03478=1050.776,-82.826,-68.807,170.144,30.797,155.829
C03479=1050.783,-82.542,-68.820,170.146,30.799,155.829
C03480=1050.789,-82.293,-68.830,170.148,30.800,155.829
C03481=1050.796,-82.043,-68.841,170.151,30.801,155.829
C03482=1050.801,-81.793,-68.852,170.153,30.802,155.829
C03483=1050.808,-81.543,-68.863,170.155,30.803,155.829
C03484=1050.814,-81.294,-68.873,170.157,30.804,155.830
C03485=1050.821,-81.044,-68.885,170.159,30.804,155.830
C03486=1050.827,-80.795,-68.896,170.161,30.805,155.830
C03487=1050.834,-80.545,-68.907,170.163,30.807,155.830
C03488=1050.839,-80.295,-68.918,170.165,30.807,155.830
C03489=1050.846,-80.045,-68.929,170.167,30.808,155.830
C03490=1050.851,-79.796,-68.940,170.169,30.809,155.830
C03491=1050.858,-79.546,-68.952,170.171,30.810,155.830
C03492=1050.864,-79.297,-68.963,170.173,30.811,155.830
C03493=1050.871,-79.047,-68.973,170.175,30.813,155.830
C03494=1050.877,-78.797,-68.984,170.177,30.814,155.830
C03495=1050.883,-78.547,-68.996,170.180,30.815,155.830
C03496=1050.889,-78.298,-69.007,170.181,30.816,155.830
C03497=1050.895,-78.048,-69.018,170.183,30.817,155.830
C03498=1050.901,-77.798,-69.029,170.185,30.818,155.830
C03499=1050.908,-77.549,-69.041,170.187,30.819,155.830
C03500=1050.913,-77.299,-69.052,170.189,30.820,155.830
C03501=1050.920,-77.049,-69.063,170.191,30.822,155.831
C03502=1050.926,-76.800,-69.074,170.194,30.823,155.831
C03503=1050.932,-76.550,-69.086,170.196,30.824,155.831
C03504=1050.938,-76.301,-69.097,170.198,30.824,155.831
C03505=1050.944,-76.050,-69.108,170.199,30.826,155.831
C03506=1050.951,-75.801,-69.120,170.201,30.827,155.831
C03507=1050.957,-75.551,-69.131,170.203,30.828,155.831
C03508=1050.963,-75.301,-69.142,170.205,30.829,155.831
C03509=1050.969,-75.052,-69.154,170.207,30.830,155.831
C03510=1050.975,-74.802,-69.165,170.210,30.831,155.831
C03511=1050.981,-74.553,-69.176,170.212,30.832,155.831
C03512=1050.988,-74.303,-69.188,170.214,30.833,155.831
C03513=1050.994,-74.053,-69.199,170.216,30.835,155.831
C03514=1051.000,-73.804,-69.211,170.218,30.836,155.832
C03515=1051.007,-73.554,-69.222,170.219,30.837,155.832
C03516=1051.013,-73.305,-69.234,170.221,30.838,155.832
C03517=1051.018,-73.054,-69.246,170.223,30.840,155.832
C03518=1051.024,-72.805,-69.256,170.225,30.841,155.832
C03519=1051.031,-72.555,-69.268,170.228,30.842,155.832
C03520=1051.036,-72.306,-69.279,170.230,30.843,155.832
C03521=1051.042,-72.056,-69.292,170.232,30.844,155.832
C03522=1051.048,-71.807,-69.303,170.234,30.846,155.832
C03523=1051.055,-71.557,-69.315,170.235,30.847,155.832
C03524=1051.061,-71.307,-69.326,170.237,30.848,155.833
C03525=1051.066,-71.058,-69.338,170.239,30.849,155.833
C03526=1051.073,-70.807,-69.349,170.241,30.851,155.833
C03527=1051.079,-70.559,-69.361,170.243,30.852,155.833
C03528=1051.085,-70.308,-69.372,170.245,30.853,155.833
C03529=1051.091,-70.058,-69.385,170.247,30.854,155.833
C03530=1051.097,-69.810,-69.396,170.250,30.856,155.833
C03531=1051.103,-69.559,-69.408,170.252,30.857,155.833
C03532=1051.109,-69.311,-69.419,170.253,30.858,155.833
C03533=1051.115,-69.060,-69.431,170.255,30.859,155.833
C03534=1051.122,-68.810,-69.443,170.257,30.861,155.834
C03535=1051.127,-68.561,-69.454,170.259,30.862,155.834
C03536=1051.134,-68.311,-69.466,170.261,30.863,155.834
C03537=1051.140,-68.062,-69.478,170.263,30.864,155.834
C03538=1051.146,-67.812,-69.489,170.265,30.866,155.834
C03539=1051.152,-67.562,-69.501,170.267,30.867,155.834
C03540=1051.159,-67.281,-69.515,170.269,30.868,155.834
C03541=1051.165,-66.998,-69.528,170.271,30.870,155.834
C03542=1051.172,-66.716,-69.541,170.273,30.871,155.834
C03543=1051.180,-66.435,-69.554,170.276,30.873,155.835
C03544=1051.186,-66.185,-69.567,170.278,30.874,155.835
C03545=1051.192,-65.935,-69.578,170.280,30.876,155.835
C03546=1051.198,-65.686,-69.589,170.282,30.877,155.835
C03547=1051.205,-65.437,-69.601,170.284,30.878,155.835
C03548=1051.210,-65.186,-69.613,170.286,30.879,155.835
C03549=1051.217,-64.937,-69.625,170.287,30.881,155.835
C03550=1051.223,-64.688,-69.637,170.289,30.882,155.835
C03551=1051.228,-64.437,-69.649,170.291,30.883,155.835
C03552=1051.235,-64.188,-69.661,170.294,30.885,155.836
C03553=1051.241,-63.939,-69.672,170.296,30.886,155.836
C03554=1051.247,-63.689,-69.685,170.298,30.887,155.836
C03555=1051.253,-63.439,-69.696,170.300,30.889,155.836
C03556=1051.260,-63.189,-69.708,170.302,30.890,155.836
C03557=1051.265,-62.940,-69.720,170.303,30.891,155.836
C03558=1051.272,-62.691,-69.732,170.305,30.892,155.836
C03559=1051.279,-62.441,-69.744,170.307,30.894,155.836
C03560=1051.284,-62.190,-69.756,170.309,30.895,155.837
C03561=1051.290,-61.942,-69.767,170.311,30.896,155.837
C03562=1051.297,-61.692,-69.779,170.313,30.898,155.837
C03563=1051.303,-61.442,-69.792,170.315,30.899,155.837
C03564=1051.310,-61.193,-69.804,170.317,30.900,155.837
C03565=1051.316,-60.942,-69.815,170.319,30.902,155.837
C03566=1051.321,-60.693,-69.827,170.321,30.903,155.837
C03567=1051.328,-60.444,-69.839,170.323,30.904,155.837
C03568=1051.334,-60.194,-69.851,170.325,30.906,155.837
C03569=1051.340,-59.944,-69.864,170.327,30.907,155.838
C03570=1051.347,-59.695,-69.876,170.329,30.908,155.838
C03571=1051.353,-59.446,-69.887,170.331,30.910,155.838
C03572=1051.359,-59.196,-69.900,170.333,30.911,155.838
C03573=1051.365,-58.946,-69.911,170.335,30.912,155.838
C03574=1051.372,-58.696,-69.923,170.336,30.914,155.838
C03575=1051.378,-58.446,-69.936,170.338,30.915,155.838
C03576=1051.385,-58.197,-69.948,170.340,30.916,155.838
C03577=1051.391,-57.948,-69.959,170.342,30.918,155.839
C03578=1051.396,-57.698,-69.972,170.344,30.919,155.839
C03579=1051.403,-57.448,-69.984,170.346,30.920,155.839
C03580=1051.409,-57.198,-69.996,170.349,30.922,155.839
C03581=1051.416,-56.949,-70.008,170.351,30.923,155.839
C03582=1051.422,-56.699,-70.020,170.352,30.924,155.839
C03583=1051.428,-56.449,-70.033,170.354,30.926,155.839
C03584=1051.435,-56.200,-70.045,170.356,30.927,155.839
C03585=1051.441,-55.950,-70.057,170.358,30.928,155.840
C03586=1051.447,-55.701,-70.069,170.360,30.930,155.840
C03587=1051.453,-55.452,-70.081,170.362,30.932,155.840
C03588=1051.459,-55.202,-70.093,170.364,30.932,155.840
C03589=1051.466,-54.952,-70.105,170.366,30.934,155.840
C03590=1051.473,-54.702,-70.117,170.368,30.936,155.840
C03591=1051.479,-54.453,-70.130,170.369,30.936,155.840
C03592=1051.485,-54.203,-70.142,170.371,30.938,155.840
C03593=1051.491,-53.953,-70.154,170.373,30.940,155.841
C03594=1051.498,-53.704,-70.166,170.375,30.941,155.841
C03595=1051.504,-53.454,-70.179,170.377,30.942,155.841
C03596=1051.510,-53.204,-70.191,170.379,30.944,155.841
C03597=1051.517,-52.955,-70.203,170.381,30.945,155.841
C03598=1051.523,-52.705,-70.216,170.383,30.947,155.841
C03599=1051.530,-52.456,-70.228,170.385,30.948,155.841
C03600=1051.536,-52.206,-70.241,170.387,30.949,155.842
C03601=1051.542,-51.956,-70.253,170.389,30.951,155.842
C03602=1051.549,-51.707,-70.264,170.391,30.952,155.842
C03603=1051.555,-51.457,-70.277,170.393,30.953,155.842
C03604=1051.562,-51.176,-70.291,170.395,30.955,155.842
C03605=1051.569,-50.896,-70.305,170.397,30.956,155.842
C03606=1051.576,-50.615,-70.319,170.400,30.958,155.842
C03607=1051.583,-50.335,-70.332,170.401,30.959,155.843
C03608=1051.590,-50.085,-70.345,170.403,30.961,155.843
C03609=1051.596,-49.835,-70.358,170.405,30.963,155.843
C03610=1051.602,-49.586,-70.370,170.407,30.964,155.843
